KUKA KRL program: MyProgram_169().src

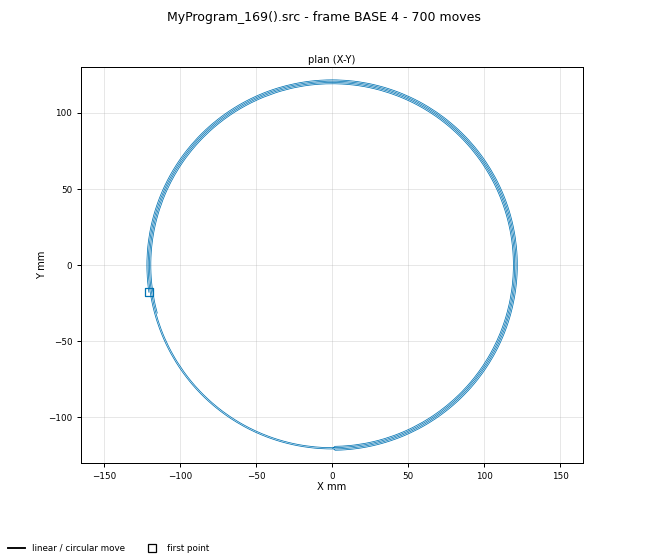
[picture p0: tool path of MyProgram_169().src in frame BASE 4, 700 of 700 moves have a stored position in this frame; points joined in program order, loops and branches not executed]
&ACCESS RVP
&REL 1
&PARAM TEMPLATE = C:\KRC\Roboter\Template\vorgabe
&PARAM EDITMASK = *
DEF MyProgram_169()
; ---- Setting reference (Base) ----
$BASE = BASE_DATA[4]

; --------------------------
; ---- Setting tool (TCP) ----
$TOOL = TOOL_DATA[3]
; --------------------------

$VEL.CP = VEL_APROX_PRINT
Startdeposition()
$VEL.CP = VEL_PRINT
LIN {X -120.4761,Y -17.8709,Z 127,A -175.5982,B 24.9546,C -1.5561,E1 24.8414,E2 261.8458} C_DIS
LIN {X -120.8784,Y -14.9089,Z 127,A -177.0141,B 24.9544,C -1.5602,E1 24.8409,E2 263.2603} C_DIS
LIN {X -121.2969,Y -10.9729,Z 127,A -178.8966,B 24.9541,C -1.5654,E1 24.8404,E2 265.1418} C_DIS
LIN {X -121.5297,Y -7.9928,Z 127,A 179.6363,B 24.954,C -1.5674,E1 24.8401,E2 266.6131} C_DIS
LIN {X -121.7415,Y -3.5142,Z 127,A 177.5701,B 24.9535,C -1.5761,E1 24.8398,E2 268.6709} C_DIS
LIN {X -121.7924,Y -0.3822,Z 127,A 176.0888,B 24.9532,C -1.5805,E1 24.8398,E2 270.1505} C_DIS
LIN {X -121.7576,Y 2.989,Z 127,A 174.4893,B 24.9529,C -1.5851,E1 24.8398,E2 271.7487} C_DIS
LIN {X -121.6476,Y 5.9762,Z 127,A 173.073,B 24.9527,C -1.5893,E1 24.84,E2 273.1637} C_DIS
LIN {X -121.479,Y 8.7426,Z 127,A 171.7841,B 24.9524,C -1.5942,E1 24.8403,E2 274.4485} C_DIS
LIN {X -121.2078,Y 11.9379,Z 127,A 170.241,B 24.9522,C -1.5977,E1 24.8407,E2 275.9927} C_DIS
LIN {X -120.7538,Y 15.8701,Z 127,A 168.3665,B 24.9518,C -1.6032,E1 24.8413,E2 277.8651} C_DIS
LIN {X -120.2477,Y 19.348,Z 127,A 166.7006,B 24.9515,C -1.6081,E1 24.842,E2 279.5294} C_DIS
LIN {X -119.8297,Y 21.776,Z 127,A 165.4749,B 24.9515,C -1.609,E1 24.8426,E2 280.7601} C_DIS
LIN {X -118.947,Y 26.1719,Z 127,A 163.3508,B 24.9511,C -1.6152,E1 24.8438,E2 282.882} C_DIS
LIN {X -118.1443,Y 29.5936,Z 127,A 161.7444,B 24.9507,C -1.6225,E1 24.8448,E2 284.4804} C_DIS
LIN {X -117.1182,Y 33.4165,Z 127,A 159.8693,B 24.9503,C -1.628,E1 24.8462,E2 286.3533} C_DIS
LIN {X -116.1073,Y 36.7826,Z 127,A 158.2044,B 24.95,C -1.6327,E1 24.8476,E2 288.0166} C_DIS
LIN {X -114.8487,Y 40.5354,Z 127,A 156.3297,B 24.9497,C -1.6381,E1 24.8493,E2 289.8892} C_DIS
LIN {X -113.8193,Y 43.3418,Z 127,A 154.914,B 24.9495,C -1.6421,E1 24.8507,E2 291.3033} C_DIS
LIN {X -112.7214,Y 46.122,Z 127,A 153.4984,B 24.9492,C -1.646,E1 24.8521,E2 292.7174} C_DIS
LIN {X -111.5555,Y 48.8744,Z 127,A 152.0828,B 24.949,C -1.65,E1 24.8537,E2 294.1314} C_DIS
LIN {X -110.3225,Y 51.5974,Z 127,A 150.6089,B 24.949,C -1.6514,E1 24.8554,E2 295.6101} C_DIS
LIN {X -108.3486,Y 55.6231,Z 127,A 148.5441,B 24.9484,C -1.6596,E1 24.858,E2 297.6663} C_DIS
LIN {X -106.7004,Y 58.7272,Z 127,A 146.8803,B 24.9481,C -1.664,E1 24.8602,E2 299.3284} C_DIS
LIN {X -104.7338,Y 62.1624,Z 127,A 144.948,B 24.948,C -1.6665,E1 24.8629,E2 301.2648} C_DIS
LIN {X -102.4536,Y 65.8526,Z 127,A 142.9275,B 24.9475,C -1.6732,E1 24.8659,E2 303.2795} C_DIS
LIN {X -100.7249,Y 68.4678,Z 127,A 141.4691,B 24.9472,C -1.6781,E1 24.8681,E2 304.7336} C_DIS
LIN {X -99.0143,Y 70.9191,Z 127,A 140.0543,B 24.947,C -1.6817,E1 24.8704,E2 306.1469} C_DIS
LIN {X -97.244,Y 73.3277,Z 127,A 138.6399,B 24.9468,C -1.6852,E1 24.8728,E2 307.5597} C_DIS
LIN {X -95.4152,Y 75.6921,Z 127,A 137.1671,B 24.9468,C -1.6861,E1 24.8753,E2 309.0373} C_DIS
LIN {X -92.5645,Y 79.1527,Z 127,A 135.1043,B 24.9462,C -1.6936,E1 24.879,E2 311.0916} C_DIS
LIN {X -90.2436,Y 81.7921,Z 127,A 133.4417,B 24.946,C -1.6975,E1 24.8821,E2 312.7526} C_DIS
LIN {X -88.4889,Y 83.6847,Z 127,A 132.2359,B 24.9458,C -1.7009,E1 24.8844,E2 313.9555} C_DIS
LIN {X -86.1216,Y 86.1216,Z 127,A 130.614,B 24.9456,C -1.7038,E1 24.8875,E2 315.5774} C_DIS
LIN {X -83.2761,Y 88.8731,Z 127,A 128.6841,B 24.9455,C -1.7053,E1 24.8915,E2 317.5116} C_DIS
LIN {X -81.07,Y 90.8901,Z 127,A 127.3051,B 24.9452,C -1.7098,E1 24.8943,E2 318.8854} C_DIS
LIN {X -78.415,Y 93.193,Z 127,A 125.6676,B 24.9449,C -1.7142,E1 24.8978,E2 320.5188} C_DIS
LIN {X -75.344,Y 95.6903,Z 127,A 123.7965,B 24.9447,C -1.718,E1 24.9018,E2 322.388} C_DIS
LIN {X -72.9729,Y 97.5105,Z 127,A 122.3839,B 24.9445,C -1.7207,E1 24.905,E2 323.7992} C_DIS
LIN {X -70.5579,Y 99.272,Z 127,A 120.913,B 24.9445,C -1.7207,E1 24.9083,E2 325.2751} C_DIS
LIN {X -67.6653,Y 101.2683,Z 127,A 119.3107,B 24.9442,C -1.7263,E1 24.912,E2 326.8696} C_DIS
LIN {X -64.3377,Y 103.4118,Z 127,A 117.4409,B 24.9439,C -1.7295,E1 24.9164,E2 328.7377} C_DIS
LIN {X -61.7805,Y 104.9596,Z 127,A 116.0291,B 24.9438,C -1.7319,E1 24.9198,E2 330.1482} C_DIS
LIN {X -59.186,Y 106.4442,Z 127,A 114.6303,B 24.9436,C -1.7347,E1 24.9232,E2 331.5444} C_DIS
LIN {X -56.5559,Y 107.8646,Z 127,A 113.2061,B 24.9435,C -1.7363,E1 24.9267,E2 332.9687} C_DIS
LIN {X -53.8918,Y 109.2201,Z 127,A 111.7368,B 24.9435,C -1.7358,E1 24.9304,E2 334.4431} C_DIS
LIN {X -50.7187,Y 110.7315,Z 127,A 110.136,B 24.9432,C -1.7407,E1 24.9344,E2 336.0363} C_DIS
LIN {X -47.986,Y 111.9428,Z 127,A 108.7252,B 24.9431,C -1.7426,E1 24.938,E2 337.446} C_DIS
LIN {X -45.2243,Y 113.0868,Z 127,A 107.3148,B 24.943,C -1.7444,E1 24.9417,E2 338.8552} C_DIS
LIN {X -42.4354,Y 114.1626,Z 127,A 105.9046,B 24.9429,C -1.7461,E1 24.9453,E2 340.2643} C_DIS
LIN {X -38.7026,Y 115.4792,Z 127,A 104.0371,B 24.9427,C -1.7482,E1 24.9503,E2 342.1304} C_DIS
LIN {X -35.355,Y 116.5499,Z 127,A 102.3796,B 24.9427,C -1.7499,E1 24.9547,E2 343.7868} C_DIS
LIN {X -32.4841,Y 117.3824,Z 127,A 100.9703,B 24.9425,C -1.7513,E1 24.9585,E2 345.1949} C_DIS
LIN {X -30.1025,Y 118.0135,Z 127,A 99.8086,B 24.9425,C -1.7524,E1 24.9616,E2 346.3558} C_DIS
LIN {X -27.0068,Y 118.7607,Z 127,A 98.3284,B 24.9423,C -1.7546,E1 24.9656,E2 347.8328} C_DIS
LIN {X -24.2756,Y 119.3484,Z 127,A 96.9905,B 24.9423,C -1.7546,E1 24.9693,E2 349.172} C_DIS
LIN {X -20.8222,Y 120.0012,Z 127,A 95.3345,B 24.9423,C -1.7558,E1 24.9738,E2 350.8271} C_DIS
LIN {X -17.8709,Y 120.4761,Z 127,A 93.9263,B 24.9422,C -1.7567,E1 24.9777,E2 352.2345} C_DIS
LIN {X -14.9089,Y 120.8784,Z 127,A 92.5183,B 24.9422,C -1.7575,E1 24.9816,E2 353.6417} C_DIS
LIN {X -10.9729,Y 121.2969,Z 127,A 90.6182,B 24.9422,C -1.7568,E1 24.9869,E2 355.5445} C_DIS
LIN {X -7.9928,Y 121.5297,Z 127,A 89.1883,B 24.9422,C -1.7563,E1 24.9909,E2 356.976} C_DIS
LIN {X -3.5142,Y 121.7415,Z 127,A 87.1351,B 24.942,C -1.7596,E1 24.9966,E2 359.0219} C_DIS
LIN {X 0,Y 121.7943,Z 127,A 85.4814,B 24.942,C -1.7599,E1 25.0012,E2 360.6749} C_DIS
LIN {X 2.989,Y 121.7576,Z 127,A 84.0744,B 24.942,C -1.76,E1 25.0051,E2 362.0813} C_DIS
LIN {X 5.9762,Y 121.6476,Z 127,A 82.668,B 24.942,C -1.76,E1 25.009,E2 363.4872} C_DIS
LIN {X 8.8861,Y 121.4693,Z 127,A 81.3102,B 24.9419,C -1.7607,E1 25.0128,E2 364.8429} C_DIS
LIN {X 11.9379,Y 121.2078,Z 127,A 79.8563,B 24.9419,C -1.7599,E1 25.0169,E2 366.2978} C_DIS
LIN {X 14.387,Y 120.9395,Z 127,A 78.6973,B 24.9419,C -1.7598,E1 25.0201,E2 367.4564} C_DIS
LIN {X 17.3507,Y 120.55,Z 127,A 77.2919,B 24.9419,C -1.7595,E1 25.024,E2 368.8613} C_DIS
LIN {X 20.5987,Y 120.0386,Z 127,A 75.7701,B 24.9419,C -1.7601,E1 25.0281,E2 370.3801} C_DIS
LIN {X 23.2449,Y 119.5534,Z 127,A 74.4816,B 24.942,C -1.7585,E1 25.0317,E2 371.6708} C_DIS
LIN {X 26.6853,Y 118.835,Z 127,A 72.8298,B 24.942,C -1.7577,E1 25.0362,E2 373.3223} C_DIS
LIN {X 30.5323,Y 117.903,Z 127,A 70.97,B 24.9422,C -1.7568,E1 25.0412,E2 375.1816} C_DIS
LIN {X 33.4165,Y 117.1182,Z 127,A 69.566,B 24.9422,C -1.7559,E1 25.045,E2 376.5855} C_DIS
LIN {X 36.7826,Y 116.1072,Z 127,A 67.9153,B 24.9422,C -1.7547,E1 25.0494,E2 378.2359} C_DIS
LIN {X 40.5354,Y 114.8487,Z 127,A 66.0565,B 24.9424,C -1.7533,E1 25.0543,E2 380.0945} C_DIS
LIN {X 43.3418,Y 113.8193,Z 127,A 64.6532,B 24.9424,C -1.7521,E1 25.058,E2 381.4977} C_DIS
LIN {X 46.122,Y 112.7214,Z 127,A 63.1921,B 24.9427,C -1.748,E1 25.0618,E2 382.965} C_DIS
LIN {X 49.0979,Y 111.4581,Z 127,A 61.7559,B 24.9426,C -1.7503,E1 25.0655,E2 384.3923} C_DIS
LIN {X 51.5974,Y 110.3225,Z 127,A 60.3866,B 24.9429,C -1.7451,E1 25.069,E2 385.7705} C_DIS
LIN {X 54.2893,Y 109.023,Z 127,A 58.9841,B 24.943,C -1.7435,E1 25.0725,E2 387.173} C_DIS
LIN {X 57.3868,Y 107.427,Z 127,A 57.4071,B 24.943,C -1.7443,E1 25.0764,E2 388.744} C_DIS
LIN {X 60.0322,Y 105.9716,Z 127,A 55.9912,B 24.943,C -1.7425,E1 25.0798,E2 390.1599} C_DIS
LIN {X 63.443,Y 103.9631,Z 127,A 54.135,B 24.9433,C -1.74,E1 25.0843,E2 392.0163} C_DIS
LIN {X 66.4175,Y 102.091,Z 127,A 52.4873,B 24.9434,C -1.7376,E1 25.0881,E2 393.6643} C_DIS
LIN {X 68.4678,Y 100.7249,Z 127,A 51.3323,B 24.9435,C -1.7359,E1 25.0908,E2 394.8194} C_DIS
LIN {X 71.3468,Y 98.7091,Z 127,A 49.6849,B 24.9437,C -1.7333,E1 25.0946,E2 396.4672} C_DIS
LIN {X 73.3277,Y 97.244,Z 127,A 48.4725,B 24.944,C -1.7287,E1 25.0973,E2 397.6862} C_DIS
LIN {X 76.1043,Y 95.0893,Z 127,A 46.8832,B 24.944,C -1.7287,E1 25.1008,E2 399.2696} C_DIS
LIN {X 78.415,Y 93.193,Z 127,A 45.4829,B 24.9442,C -1.7262,E1 25.1038,E2 400.6703} C_DIS
LIN {X 80.4881,Y 91.4068,Z 127,A 44.2246,B 24.9442,C -1.7251,E1 25.1064,E2 401.9263} C_DIS
LIN {X 82.8933,Y 89.2331,Z 127,A 42.6826,B 24.9445,C -1.7211,E1 25.1096,E2 403.4715} C_DIS
LIN {X 85.0583,Y 87.1719,Z 127,A 41.283,B 24.9447,C -1.7184,E1 25.1124,E2 404.8716} C_DIS
LIN {X 88.2092,Y 83.9821,Z 127,A 39.1831,B 24.9449,C -1.7142,E1 25.1165,E2 406.9724} C_DIS
LIN {X 90.1788,Y 81.8627,Z 127,A 37.8259,B 24.9451,C -1.7113,E1 25.1191,E2 408.3304} C_DIS
LIN {X 92.2237,Y 79.5527,Z 127,A 36.3843,B 24.9453,C -1.7084,E1 25.1217,E2 409.7724} C_DIS
LIN {X 93.9,Y 77.5642,Z 127,A 35.1835,B 24.9454,C -1.7066,E1 25.1239,E2 410.9719} C_DIS
LIN {X 96.0161,Y 74.9317,Z 127,A 33.5862,B 24.9457,C -1.7023,E1 25.1267,E2 412.5718} C_DIS
LIN {X 97.8261,Y 72.5528,Z 127,A 32.1876,B 24.9459,C -1.6992,E1 25.129,E2 413.9712} C_DIS
LIN {X 99.5772,Y 70.1302,Z 127,A 30.7889,B 24.9461,C -1.696,E1 25.1313,E2 415.3707} C_DIS
LIN {X 101.2683,Y 67.6653,Z 127,A 29.3903,B 24.9463,C -1.6927,E1 25.1335,E2 416.77} C_DIS
LIN {X 102.8984,Y 65.1597,Z 127,A 27.9919,B 24.9465,C -1.6894,E1 25.1356,E2 418.1694} C_DIS
LIN {X 104.1936,Y 63.0638,Z 127,A 26.8099,B 24.9468,C -1.6852,E1 25.1373,E2 419.3552} C_DIS
LIN {X 105.9716,Y 60.0322,Z 127,A 25.1958,B 24.9469,C -1.6826,E1 25.1396,E2 420.9672} C_DIS
LIN {X 107.1624,Y 57.8753,Z 127,A 23.9859,B 24.9473,C -1.6769,E1 25.1412,E2 422.1841} C_DIS
LIN {X 108.7896,Y 54.7601,Z 127,A 22.4,B 24.9473,C -1.6755,E1 25.1432,E2 423.7648} C_DIS
LIN {X 110.5097,Y 51.1951,Z 127,A 20.549,B 24.9477,C -1.6708,E1 25.1454,E2 425.617} C_DIS
LIN {X 111.9428,Y 47.986,Z 127,A 18.9056,B 24.948,C -1.6664,E1 25.1473,E2 427.2618} C_DIS
LIN {X 113.0047,Y 45.4259,Z 127,A 17.6339,B 24.9481,C -1.6642,E1 25.1486,E2 428.5317} C_DIS
LIN {X 114.1626,Y 42.4354,Z 127,A 16.1111,B 24.9484,C -1.659,E1 25.1501,E2 430.0583} C_DIS
LIN {X 115.4792,Y 38.7026,Z 127,A 14.2361,B 24.9488,C -1.6527,E1 25.1519,E2 431.9375} C_DIS
LIN {X 116.5499,Y 35.355,Z 127,A 12.618,B 24.949,C -1.6494,E1 25.1532,E2 433.5543} C_DIS
LIN {X 117.3824,Y 32.4841,Z 127,A 11.2212,B 24.9493,C -1.6455,E1 25.1543,E2 434.9522} C_DIS
LIN {X 118.374,Y 28.6521,Z 127,A 9.3711,B 24.9496,C -1.6403,E1 25.1555,E2 436.8038} C_DIS
LIN {X 119.1535,Y 25.225,Z 127,A 7.7291,B 24.9499,C -1.6356,E1 25.1565,E2 438.4474} C_DIS
LIN {X 120.0012,Y 20.8222,Z 127,A 5.6337,B 24.9502,C -1.6296,E1 25.1576,E2 440.5447} C_DIS
LIN {X 120.4761,Y 17.8709,Z 127,A 4.2371,B 24.9505,C -1.6256,E1 25.1582,E2 441.9425} C_DIS
LIN {X 120.8784,Y 14.9089,Z 127,A 2.8405,B 24.9507,C -1.6216,E1 25.1587,E2 443.3404} C_DIS
LIN {X 121.1531,Y 12.4605,Z 127,A 1.6525,B 24.951,C -1.6164,E1 25.1591,E2 444.5336} C_DIS
LIN {X 121.4643,Y 8.9597,Z 127,A 0.047,B 24.9512,C -1.6134,E1 25.1594,E2 446.1366} C_DIS
LIN {X 121.6476,Y 5.9762,Z 127,A -1.3495,B 24.9515,C -1.6093,E1 25.1596,E2 447.5344} C_DIS
LIN {X 121.7576,Y 2.989,Z 127,A -2.746,B 24.9517,C -1.6052,E1 25.1598,E2 448.9323} C_DIS
LIN {X 121.7924,Y -0.3822,Z 127,A -4.1792,B 24.9516,C -1.6077,E1 25.1598,E2 450.3511} C_DIS
LIN {X 121.7576,Y -2.989,Z 127,A -5.5389,B 24.9522,C -1.597,E1 25.1598,E2 451.728} C_DIS
LIN {X 121.6476,Y -5.9762,Z 127,A -6.9354,B 24.9525,C -1.5928,E1 25.1595,E2 453.126} C_DIS
LIN {X 121.4643,Y -8.9597,Z 127,A -8.3318,B 24.9527,C -1.5887,E1 25.1593,E2 454.5238} C_DIS
LIN {X 121.2078,Y -11.9379,Z 127,A -9.728,B 24.953,C -1.5846,E1 25.1589,E2 455.9215} C_DIS
LIN {X 120.7538,Y -15.8701,Z 127,A -11.6351,B 24.9534,C -1.5763,E1 25.1583,E2 457.8368} C_DIS
LIN {X 120.328,Y -18.8287,Z 127,A -13.0315,B 24.9537,C -1.5722,E1 25.1577,E2 459.2347} C_DIS
LIN {X 119.8297,Y -21.776,Z 127,A -14.428,B 24.9539,C -1.5681,E1 25.157,E2 460.6327} C_DIS
LIN {X 119.2217,Y -24.8928,Z 127,A -15.8805,B 24.9541,C -1.5653,E1 25.1562,E2 462.0833} C_DIS
LIN {X 118.6168,Y -27.6296,Z 127,A -17.2211,B 24.9544,C -1.5599,E1 25.1554,E2 463.4288} C_DIS
LIN {X 117.5195,Y -31.9768,Z 127,A -19.2586,B 24.9546,C -1.5567,E1 25.154,E2 465.4621} C_DIS
LIN {X 116.6993,Y -34.8513,Z 127,A -20.6555,B 24.9548,C -1.5527,E1 25.1529,E2 466.8605} C_DIS
LIN {X 115.8089,Y -37.7047,Z 127,A -22.1095,B 24.9552,C -1.5458,E1 25.1516,E2 468.3225} C_DIS
LIN {X 114.6747,Y -41.0313,Z 127,A -23.6945,B 24.9553,C -1.5439,E1 25.1502,E2 469.903} C_DIS
LIN {X 113.1249,Y -45.1272,Z 127,A -25.7238,B 24.9556,C -1.539,E1 25.1481,E2 471.9325} C_DIS
LIN {X 112.1469,Y -47.5018,Z 127,A -26.9413,B 24.9559,C -1.5348,E1 25.1468,E2 473.1532} C_DIS
LIN {X 110.7315,Y -50.7188,Z 127,A -28.5838,B 24.9561,C -1.5302,E1 25.1449,E2 474.7976} C_DIS
LIN {X 109.023,Y -54.2893,Z 127,A -30.4342,B 24.9564,C -1.5252,E1 25.1427,E2 476.65} C_DIS
LIN {X 107.413,Y -57.4134,Z 127,A -32.0769,B 24.9567,C -1.5207,E1 25.1406,E2 478.2945} C_DIS
LIN {X 105.9716,Y -60.0322,Z 127,A -33.4742,B 24.9569,C -1.517,E1 25.1387,E2 479.6934} C_DIS
LIN {X 104.4665,Y -62.6148,Z 127,A -34.8717,B 24.9571,C -1.5133,E1 25.1367,E2 481.0924} C_DIS
LIN {X 103.1304,Y -64.7883,Z 127,A -36.1065,B 24.9574,C -1.5081,E1 25.1348,E2 482.3331} C_DIS
LIN {X 100.7249,Y -68.4678,Z 127,A -38.1778,B 24.9577,C -1.5021,E1 25.1316,E2 484.4084} C_DIS
LIN {X 98.7091,Y -71.3468,Z 127,A -39.7641,B 24.9578,C -1.5007,E1 25.1291,E2 485.9901} C_DIS
LIN {X 96.0161,Y -74.9317,Z 127,A -41.861,B 24.9581,C -1.4956,E1 25.1255,E2 488.0893} C_DIS
LIN {X 94.1483,Y -77.2655,Z 127,A -43.2591,B 24.9583,C -1.4922,E1 25.1231,E2 489.4888} C_DIS
LIN {X 91.5862,Y -80.2827,Z 127,A -45.1686,B 24.9587,C -1.485,E1 25.1196,E2 491.4067} C_DIS
LIN {X 89.5884,Y -82.5062,Z 127,A -46.5672,B 24.9589,C -1.4817,E1 25.1169,E2 492.8068} C_DIS
LIN {X 86.4909,Y -85.7477,Z 127,A -48.6653,B 24.9591,C -1.477,E1 25.1129,E2 494.907} C_DIS
LIN {X 83.9821,Y -88.2092,Z 127,A -50.2525,B 24.9591,C -1.4762,E1 25.1097,E2 496.4895} C_DIS
LIN {X 81.7921,Y -90.2436,Z 127,A -51.6517,B 24.9593,C -1.4732,E1 25.1068,E2 497.8902} C_DIS
LIN {X 79.5527,Y -92.2237,Z 127,A -53.0511,B 24.9595,C -1.4702,E1 25.1039,E2 499.2909} C_DIS
LIN {X 76.5182,Y -94.7539,Z 127,A -54.902,B 24.9597,C -1.4665,E1 25.0999,E2 501.1437} C_DIS
LIN {X 74.164,Y -96.6077,Z 127,A -56.3617,B 24.96,C -1.4609,E1 25.0966,E2 502.6111} C_DIS
LIN {X 71.3468,Y -98.7091,Z 127,A -57.9498,B 24.96,C -1.4606,E1 25.0931,E2 504.1944} C_DIS
LIN {X 67.6925,Y -101.2499,Z 127,A -60.0261,B 24.9602,C -1.4571,E1 25.0883,E2 506.2717} C_DIS
LIN {X 64.3377,Y -103.4118,Z 127,A -61.9047,B 24.9604,C -1.4535,E1 25.0839,E2 508.1529} C_DIS
LIN {X 61.7805,Y -104.9596,Z 127,A -63.3053,B 24.9606,C -1.4511,E1 25.0805,E2 509.5548} C_DIS
LIN {X 59.186,Y -106.4442,Z 127,A -64.7638,B 24.9608,C -1.446,E1 25.0769,E2 511.021} C_DIS
LIN {X 56.5559,Y -107.8646,Z 127,A -66.1647,B 24.9609,C -1.4438,E1 25.0735,E2 512.4231} C_DIS
LIN {X 53.421,Y -109.4534,Z 127,A -67.7546,B 24.9609,C -1.4441,E1 25.0695,E2 514.008} C_DIS
LIN {X 51.1951,Y -110.5097,Z 127,A -68.9098,B 24.961,C -1.4425,E1 25.0666,E2 515.1641} C_DIS
LIN {X 47.986,Y -111.9428,Z 127,A -70.5579,B 24.9611,C -1.4402,E1 25.0624,E2 516.8137} C_DIS
LIN {X 45.3148,Y -113.0499,Z 127,A -71.8974,B 24.9611,C -1.4392,E1 25.0589,E2 518.1523} C_DIS
LIN {X 42.4354,Y -114.1626,Z 127,A -73.3617,B 24.9613,C -1.4366,E1 25.0551,E2 519.6197} C_DIS
LIN {X 38.7026,Y -115.4792,Z 127,A -75.2768,B 24.9616,C -1.4317,E1 25.05,E2 521.5426} C_DIS
LIN {X 35.355,Y -116.5499,Z 127,A -76.8683,B 24.9616,C -1.4326,E1 25.0458,E2 523.1289} C_DIS
LIN {X 32.4841,Y -117.3824,Z 127,A -78.271,B 24.9616,C -1.4312,E1 25.042,E2 524.5326} C_DIS
LIN {X 29.5936,Y -118.1443,Z 127,A -79.6742,B 24.9616,C -1.4299,E1 25.0382,E2 525.9368} C_DIS
LIN {X 26.6853,Y -118.835,Z 127,A -81.0777,B 24.9618,C -1.4287,E1 25.0344,E2 527.3412} C_DIS
LIN {X 22.8092,Y -119.6373,Z 127,A -82.9731,B 24.9619,C -1.4255,E1 25.0292,E2 529.2419} C_DIS
LIN {X 19.8663,Y -120.161,Z 127,A -84.3981,B 24.962,C -1.4235,E1 25.0253,E2 530.6701} C_DIS
LIN {X 16.9114,Y -120.6124,Z 127,A -85.8021,B 24.962,C -1.4226,E1 25.0214,E2 532.075} C_DIS
LIN {X 13.4321,Y -121.0513,Z 127,A -87.3904,B 24.962,C -1.4245,E1 25.017,E2 533.6576} C_DIS
LIN {X 8.9597,Y -121.4643,Z 127,A -89.5027,B 24.962,C -1.4234,E1 25.0111,E2 535.7713} C_DIS
LIN {X 5.9762,Y -121.6476,Z 127,A -90.9077,B 24.962,C -1.4229,E1 25.0072,E2 537.177} C_DIS
LIN {X 2.02,Y -121.7755,Z 127,A -92.7723,B 24.9621,C -1.4222,E1 25.002,E2 539.0428} C_DIS
LIN {X 2.02,Y -121.7755,Z 127,A -92.7723,B 24.9621,C -1.4222,E1 25.002,E2 539.0428} C_DIS
Enddeposition()
LIN {X 0.8498,Y -120.9267,Z 127,A -92.499,B 24.9592,C -1.476,E1 25.0031,E2 538.6421} C_DIS
Startdeposition()
$VEL.CP = VEL_PRINT
LIN {X 6.1613,Y -120.7806,Z 127,A -89.7657,B 24.9586,C -1.4871,E1 25.0108,E2 535.8835} C_DIS
LIN {X 9.6002,Y -120.5549,Z 127,A -88.5598,B 24.9597,C -1.4675,E1 25.014,E2 534.7243} C_DIS
LIN {X 12.7244,Y -120.2653,Z 127,A -87.0113,B 24.9594,C -1.4713,E1 25.0183,E2 533.168} C_DIS
LIN {X 17.3332,Y -119.6884,Z 127,A -84.2229,B 24.9578,C -1.501,E1 25.0263,E2 530.3116} C_DIS
LIN {X 21.9078,Y -118.9368,Z 127,A -82.5343,B 24.9591,C -1.4783,E1 25.0307,E2 528.6786} C_DIS
LIN {X 25.5115,Y -118.2154,Z 127,A -80.9082,B 24.9593,C -1.4744,E1 25.0352,E2 527.0639} C_DIS
LIN {X 28.6124,Y -117.5031,Z 127,A -79.4189,B 24.9593,C -1.475,E1 25.0392,E2 525.5753} C_DIS
LIN {X 32.2121,Y -116.5698,Z 127,A -77.5756,B 24.9589,C -1.4807,E1 25.0442,E2 523.7212} C_DIS
LIN {X 35.1312,Y -115.7236,Z 127,A -75.4821,B 24.957,C -1.5142,E1 25.05,E2 521.5524} C_DIS
LIN {X 39.9144,Y -114.16,Z 127,A -73.194,B 24.9571,C -1.5126,E1 25.056,E2 519.2726} C_DIS
LIN {X 44.3276,Y -112.5199,Z 127,A -71.8403,B 24.9594,C -1.473,E1 25.0593,E2 518.0154} C_DIS
LIN {X 47.9828,Y -111.011,Z 127,A -69.6996,B 24.9585,C -1.4887,E1 25.0649,E2 515.8427} C_DIS
LIN {X 51.186,Y -109.5704,Z 127,A -68.0535,B 24.9584,C -1.4905,E1 25.069,E2 514.1965} C_DIS
LIN {X 54.5225,Y -107.9503,Z 127,A -66.317,B 24.9583,C -1.4924,E1 25.0734,E2 512.4602} C_DIS
LIN {X 58.0159,Y -106.1129,Z 127,A -64.4585,B 24.9581,C -1.4951,E1 25.078,E2 510.6006} C_DIS
LIN {X 61.2525,Y -104.2779,Z 127,A -62.6716,B 24.9579,C -1.4995,E1 25.0823,E2 508.8086} C_DIS
LIN {X 64.1573,Y -102.5158,Z 127,A -61.0731,B 24.9577,C -1.5021,E1 25.0861,E2 507.2092} C_DIS
LIN {X 67.5687,Y -100.3005,Z 127,A -59.3271,B 24.958,C -1.497,E1 25.0901,E2 505.4808} C_DIS
LIN {X 72.1717,Y -97.0424,Z 127,A -56.1531,B 24.9563,C -1.5273,E1 25.0975,E2 502.2464} C_DIS
LIN {X 74.8604,Y -94.982,Z 127,A -54.9366,B 24.9572,C -1.5117,E1 25.1,E2 501.0714} C_DIS
LIN {X 79.4487,Y -91.1788,Z 127,A -52.0227,B 24.9566,C -1.5226,E1 25.1063,E2 498.143} C_DIS
LIN {X 82.7863,Y -88.1594,Z 127,A -49.946,B 24.9564,C -1.5249,E1 25.1105,E2 496.0692} C_DIS
LIN {X 86.0248,Y -85.0023,Z 127,A -47.4355,B 24.9551,C -1.5485,E1 25.1156,E2 493.5136} C_DIS
LIN {X 88.6717,Y -82.2391,Z 127,A -45.9364,B 24.9557,C -1.5375,E1 25.1184,E2 492.0473} C_DIS
LIN {X 93.5426,Y -76.6541,Z 127,A -42.6577,B 24.9558,C -1.5351,E1 25.1243,E2 488.789} C_DIS
LIN {X 97.9667,Y -70.9126,Z 127,A -39.0659,B 24.9549,C -1.5523,E1 25.1304,E2 485.1736} C_DIS
LIN {X 100.0389,Y -67.9551,Z 127,A -37.4767,B 24.9549,C -1.5511,E1 25.1329,E2 483.5951} C_DIS
LIN {X 101.5025,Y -65.7505,Z 127,A -36.05,B 24.9542,C -1.5633,E1 25.1351,E2 482.1468} C_DIS
LIN {X 103.9195,Y -61.8589,Z 127,A -34.0196,B 24.9542,C -1.5626,E1 25.1381,E2 480.1283} C_DIS
LIN {X 106.0589,Y -58.1155,Z 127,A -31.8672,B 24.9536,C -1.5742,E1 25.141,E2 477.9599} C_DIS
LIN {X 108.128,Y -54.1687,Z 127,A -29.947,B 24.9538,C -1.571,E1 25.1434,E2 476.0575} C_DIS
LIN {X 109.5966,Y -51.1295,Z 127,A -27.6686,B 24.9514,C -1.6101,E1 25.1462,E2 473.6991} C_DIS
LIN {X 111.5748,Y -46.6565,Z 127,A -25.9265,B 24.9527,C -1.5882,E1 25.1481,E2 472.0181} C_DIS
LIN {X 112.8287,Y -43.5406,Z 127,A -24.3633,B 24.9525,C -1.5918,E1 25.1496,E2 470.4552} C_DIS
LIN {X 114.2091,Y -39.7745,Z 127,A -22.5326,B 24.9524,C -1.5943,E1 25.1514,E2 468.6289} C_DIS
LIN {X 115.4976,Y -35.8602,Z 127,A -20.7468,B 24.9525,C -1.5921,E1 25.1529,E2 466.8583} C_DIS
LIN {X 116.2006,Y -33.517,Z 127,A -19.5938,B 24.9523,C -1.5955,E1 25.1538,E2 465.7038} C_DIS
LIN {X 117.0607,Y -30.373,Z 127,A -17.9082,B 24.9516,C -1.6076,E1 25.155,E2 463.9995} C_DIS
LIN {X 118.0996,Y -26.0426,Z 127,A -15.8721,B 24.9514,C -1.6107,E1 25.1563,E2 461.9678} C_DIS
LIN {X 118.6259,Y -23.5373,Z 127,A -14.12,B 24.9495,C -1.6419,E1 25.1573,E2 460.1525} C_DIS
LIN {X 119.3576,Y -19.4841,Z 127,A -11.8288,B 24.948,C -1.6655,E1 25.1583,E2 457.819} C_DIS
LIN {X 120.1583,Y -13.7026,Z 127,A -10.204,B 24.951,C -1.6169,E1 25.1588,E2 456.3184} C_DIS
LIN {X 120.6907,Y -7.719,Z 127,A -7.1986,B 24.95,C -1.6342,E1 25.1595,E2 453.2902} C_DIS
LIN {X 120.9156,Y -2.2507,Z 127,A -4.5831,B 24.9494,C -1.6438,E1 25.1598,E2 450.6676} C_DIS
LIN {X 120.9326,Y 1.0405,Z 127,A -2.6111,B 24.9478,C -1.6697,E1 25.1598,E2 448.6463} C_DIS
LIN {X 120.8476,Y 4.667,Z 127,A -1.4404,B 24.9491,C -1.6477,E1 25.1596,E2 447.5344} C_DIS
LIN {X 120.5298,Y 9.9136,Z 127,A 1.0724,B 24.9486,C -1.6569,E1 25.1592,E2 445.0148} C_DIS
LIN {X 119.835,Y 16.3014,Z 127,A 4.1713,B 24.9478,C -1.6694,E1 25.1582,E2 441.9049} C_DIS
LIN {X 119.3699,Y 19.4104,Z 127,A 5.7343,B 24.9472,C -1.6778,E1 25.1575,E2 440.3311} C_DIS
LIN {X 118.7629,Y 22.8257,Z 127,A 7.3217,B 24.9471,C -1.6803,E1 25.1567,E2 438.7472} C_DIS
LIN {X 117.9466,Y 26.7299,Z 127,A 9.2263,B 24.9467,C -1.6869,E1 25.1556,E2 436.8379} C_DIS
LIN {X 117.1848,Y 29.8899,Z 127,A 10.7456,B 24.9464,C -1.6907,E1 25.1545,E2 435.3185} C_DIS
LIN {X 116.1336,Y 33.7502,Z 127,A 12.6999,B 24.9459,C -1.6995,E1 25.153,E2 433.3547} C_DIS
LIN {X 115.0004,Y 37.4246,Z 127,A 14.4424,B 24.9458,C -1.7011,E1 25.1516,E2 431.6182} C_DIS
LIN {X 113.6967,Y 41.2159,Z 127,A 16.6118,B 24.9445,C -1.7203,E1 25.1495,E2 429.4158} C_DIS
LIN {X 111.8909,Y 45.8932,Z 127,A 18.6954,B 24.945,C -1.7128,E1 25.1474,E2 427.3614} C_DIS
LIN {X 110.4039,Y 49.3635,Z 127,A 20.411,B 24.945,C -1.7144,E1 25.1455,E2 425.6515} C_DIS
LIN {X 109.2523,Y 51.8642,Z 127,A 21.8103,B 24.9444,C -1.7228,E1 25.1438,E2 424.2398} C_DIS
LIN {X 107.7678,Y 54.8796,Z 127,A 23.3515,B 24.9442,C -1.7248,E1 25.1419,E2 422.7021} C_DIS
LIN {X 106.0644,Y 58.1054,Z 127,A 25.0874,B 24.9439,C -1.73,E1 25.1396,E2 420.9631} C_DIS
LIN {X 104.2158,Y 61.3576,Z 127,A 26.7893,B 24.9439,C -1.7314,E1 25.1372,E2 419.2668} C_DIS
LIN {X 102.089,Y 64.8369,Z 127,A 28.7704,B 24.9433,C -1.7389,E1 25.1343,E2 417.2779} C_DIS
LIN {X 100.502,Y 67.2711,Z 127,A 30.1844,B 24.943,C -1.7443,E1 25.1321,E2 415.8581} C_DIS
LIN {X 98.455,Y 70.2301,Z 127,A 31.6473,B 24.9435,C -1.7368,E1 25.1298,E2 414.4201} C_DIS
LIN {X 97.0709,Y 72.1337,Z 127,A 32.9753,B 24.9426,C -1.7501,E1 25.1275,E2 413.0672} C_DIS
LIN {X 94.663,Y 75.264,Z 127,A 34.7079,B 24.9427,C -1.7479,E1 25.1246,E2 411.348} C_DIS
LIN {X 92.3646,Y 78.0682,Z 127,A 36.3955,B 24.9426,C -1.7505,E1 25.1215,E2 409.662} C_DIS
LIN {X 90.1956,Y 80.5632,Z 127,A 37.9504,B 24.9424,C -1.7536,E1 25.1187,E2 408.1067} C_DIS
LIN {X 88.5364,Y 82.3854,Z 127,A 39.288,B 24.9416,C -1.7645,E1 25.1161,E2 406.7493} C_DIS
LIN {X 85.9766,Y 85.051,Z 127,A 40.9605,B 24.9416,C -1.7645,E1 25.1128,E2 405.0838} C_DIS
LIN {X 83.1235,Y 87.8423,Z 127,A 42.6587,B 24.942,C -1.7592,E1 25.1095,E2 403.4054} C_DIS
LIN {X 80.9968,Y 89.8073,Z 127,A 44.1581,B 24.9414,C -1.7682,E1 25.1064,E2 401.8907} C_DIS
LIN {X 78.6782,Y 91.8449,Z 127,A 45.599,B 24.9413,C -1.77,E1 25.1033,E2 400.4511} C_DIS
LIN {X 76.6329,Y 93.5598,Z 127,A 46.9868,B 24.9407,C -1.7784,E1 25.1003,E2 399.0488} C_DIS
LIN {X 73.8027,Y 95.8061,Z 127,A 48.5642,B 24.9409,C -1.7751,E1 25.0969,E2 397.485} C_DIS
LIN {X 70.9675,Y 97.9266,Z 127,A 50.2179,B 24.9409,C -1.7769,E1 25.0931,E2 395.8329} C_DIS
LIN {X 67.925,Y 100.0593,Z 127,A 52.1049,B 24.9402,C -1.786,E1 25.0888,E2 393.9309} C_DIS
LIN {X 64.2994,Y 102.427,Z 127,A 54.2022,B 24.9398,C -1.7915,E1 25.0838,E2 391.8275} C_DIS
LIN {X 60.2122,Y 104.8815,Z 127,A 56.4074,B 24.9398,C -1.7923,E1 25.0785,E2 389.6272} C_DIS
LIN {X 56.6016,Y 106.8737,Z 127,A 58.1264,B 24.9404,C -1.7838,E1 25.0744,E2 387.9332} C_DIS
LIN {X 53.9827,Y 108.2201,Z 127,A 59.7187,B 24.9396,C -1.795,E1 25.0703,E2 386.3188} C_DIS
LIN {X 50.3391,Y 109.9642,Z 127,A 61.7007,B 24.9392,C -1.8005,E1 25.0653,E2 384.3287} C_DIS
LIN {X 47.5957,Y 111.1789,Z 127,A 63.2415,B 24.9387,C -1.8078,E1 25.0613,E2 382.7745} C_DIS
LIN {X 43.7491,Y 112.7471,Z 127,A 64.9546,B 24.9394,C -1.7977,E1 25.0569,E2 381.0891} C_DIS
LIN {X 40.1869,Y 114.0643,Z 127,A 66.7141,B 24.9394,C -1.7975,E1 25.0523,E2 379.3337} C_DIS
LIN {X 37.2453,Y 115.0584,Z 127,A 68.179,B 24.9394,C -1.7984,E1 25.0484,E2 377.8694} C_DIS
LIN {X 33.468,Y 116.2145,Z 127,A 70.1224,B 24.9391,C -1.8032,E1 25.0432,E2 375.9181} C_DIS
LIN {X 30.0427,Y 117.1456,Z 127,A 71.7414,B 24.9391,C -1.8013,E1 25.0389,E2 374.306} C_DIS
LIN {X 26.4728,Y 118.0057,Z 127,A 73.585,B 24.9388,C -1.8071,E1 25.0338,E2 372.4512} C_DIS
LIN {X 23.0384,Y 118.722,Z 127,A 75.1383,B 24.9391,C -1.8028,E1 25.0296,E2 370.9101} C_DIS
LIN {X 19.8165,Y 119.302,Z 127,A 76.6984,B 24.9391,C -1.8038,E1 25.0253,E2 369.3492} C_DIS
LIN {X 15.97,Y 119.8782,Z 127,A 78.4708,B 24.9392,C -1.801,E1 25.0204,E2 367.585} C_DIS
LIN {X 9.6785,Y 120.5486,Z 127,A 81.3504,B 24.9395,C -1.7959,E1 25.0125,E2 364.7194} C_DIS
LIN {X 3.0343,Y 120.9003,Z 127,A 85.5678,B 24.9362,C -1.8451,E1 25.0004,E2 360.3864} C_DIS
LIN {X -2.7347,Y 120.9067,Z 127,A 87.2646,B 24.9395,C -1.7964,E1 24.996,E2 358.8049} C_DIS
LIN {X -9.5192,Y 120.5614,Z 127,A 91.6154,B 24.936,C -1.8473,E1 24.9835,E2 354.3319} C_DIS
LIN {X -15.7161,Y 119.9111,Z 127,A 93.543,B 24.9394,C -1.7984,E1 24.9785,E2 352.519} C_DIS
LIN {X -19.3379,Y 119.382,Z 127,A 95.2416,B 24.9396,C -1.7956,E1 24.9738,E2 350.8256} C_DIS
LIN {X -22.6027,Y 118.8059,Z 127,A 96.9772,B 24.9391,C -1.8019,E1 24.969,E2 349.0734} C_DIS
LIN {X -26.5397,Y 117.9906,Z 127,A 98.864,B 24.9393,C -1.7993,E1 24.9639,E2 347.1903} C_DIS
LIN {X -30.0117,Y 117.1535,Z 127,A 100.5008,B 24.9396,C -1.7952,E1 24.9594,E2 345.5609} C_DIS
LIN {X -33.0344,Y 116.3373,Z 127,A 102.0984,B 24.9394,C -1.7988,E1 24.9551,E2 343.9524} C_DIS
LIN {X -37.0774,Y 115.1127,Z 127,A 104.0442,B 24.9397,C -1.794,E1 24.9499,E2 342.0146} C_DIS
LIN {X -41.0063,Y 113.7732,Z 127,A 105.9677,B 24.94,C -1.7895,E1 24.9449,E2 340.0978} C_DIS
LIN {X -45.4273,Y 112.0805,Z 127,A 108.2574,B 24.94,C -1.7886,E1 24.9389,E2 337.8055} C_DIS
LIN {X -48.5043,Y 110.7836,Z 127,A 109.8855,B 24.94,C -1.7883,E1 24.9348,E2 336.1743} C_DIS
LIN {X -52.1558,Y 109.1122,Z 127,A 111.6745,B 24.9406,C -1.7803,E1 24.9303,E2 334.3998} C_DIS
LIN {X -54.7166,Y 107.8511,Z 127,A 113.092,B 24.9406,C -1.781,E1 24.9267,E2 332.977} C_DIS
LIN {X -57.6486,Y 106.3122,Z 127,A 114.6574,B 24.9407,C -1.7781,E1 24.9229,E2 331.4139} C_DIS
LIN {X -60.9415,Y 104.4618,Z 127,A 116.7107,B 24.9402,C -1.7866,E1 24.9178,E2 329.3344} C_DIS
LIN {X -65.1983,Y 101.857,Z 127,A 118.8485,B 24.9411,C -1.7721,E1 24.9128,E2 327.2244} C_DIS
LIN {X -67.9625,Y 100.0339,Z 127,A 120.6368,B 24.9407,C -1.7787,E1 24.9086,E2 325.4144} C_DIS
LIN {X -71.7394,Y 97.3614,Z 127,A 122.6236,B 24.9416,C -1.7651,E1 24.9042,E2 323.453} C_DIS
LIN {X -74.421,Y 95.3293,Z 127,A 124.3751,B 24.9414,C -1.7685,E1 24.9003,E2 321.687} C_DIS
LIN {X -77.6218,Y 92.7399,Z 127,A 126.1945,B 24.942,C -1.7584,E1 24.8964,E2 319.8846} C_DIS
LIN {X -80.4222,Y 90.3217,Z 127,A 128.027,B 24.942,C -1.7579,E1 24.8926,E2 318.0462} C_DIS
LIN {X -83.3447,Y 87.6343,Z 127,A 129.8636,B 24.9425,C -1.7515,E1 24.8888,E2 316.2174} C_DIS
LIN {X -85.7843,Y 85.2457,Z 127,A 131.4557,B 24.9428,C -1.7464,E1 24.8857,E2 314.6306} C_DIS
LIN {X -88.5346,Y 82.3873,Z 127,A 133.4588,B 24.9428,C -1.7471,E1 24.8818,E2 312.6172} C_DIS
LIN {X -90.875,Y 79.7965,Z 127,A 135.0148,B 24.9434,C -1.7386,E1 24.879,E2 311.0745} C_DIS
LIN {X -93.7862,Y 76.3535,Z 127,A 137.18,B 24.9436,C -1.7342,E1 24.8751,E2 308.9097} C_DIS
LIN {X -97.0149,Y 72.2083,Z 127,A 139.7397,B 24.9439,C -1.7305,E1 24.8707,E2 306.3467} C_DIS
LIN {X -99.7031,Y 68.4499,Z 127,A 141.9635,B 24.9442,C -1.7259,E1 24.8672,E2 304.123} C_DIS
LIN {X -101.7806,Y 65.3173,Z 127,A 143.6666,B 24.9447,C -1.7175,E1 24.8646,E2 302.4313} C_DIS
LIN {X -103.748,Y 62.1489,Z 127,A 145.4783,B 24.9449,C -1.7143,E1 24.862,E2 300.6179} C_DIS
LIN {X -106.8082,Y 56.7259,Z 127,A 148.3658,B 24.9457,C -1.7028,E1 24.8581,E2 297.7425} C_DIS
LIN {X -108.3525,Y 53.7158,Z 127,A 150.3976,B 24.9448,C -1.7166,E1 24.8555,E2 295.667} C_DIS
LIN {X -109.9183,Y 50.4385,Z 127,A 151.8609,B 24.9458,C -1.7002,E1 24.8538,E2 294.2349} C_DIS
LIN {X -111.5018,Y 46.8296,Z 127,A 153.6351,B 24.9464,C -1.6904,E1 24.8519,E2 292.474} C_DIS
LIN {X -112.4659,Y 44.4649,Z 127,A 155.4424,B 24.945,C -1.7125,E1 24.85,E2 290.6039} C_DIS
LIN {X -114.0449,Y 40.2422,Z 127,A 156.86,B 24.9474,C -1.6747,E1 24.8487,E2 289.2684} C_DIS
LIN {X -114.9616,Y 37.5443,Z 127,A 158.3935,B 24.9472,C -1.6783,E1 24.8473,E2 287.7175} C_DIS
LIN {X -116.1031,Y 33.8531,Z 127,A 160.336,B 24.9472,C -1.6773,E1 24.8458,E2 285.7663} C_DIS
LIN {X -117.2008,Y 29.8276,Z 127,A 162.2311,B 24.9479,C -1.6675,E1 24.8444,E2 283.8836} C_DIS
LIN {X -118.0727,Y 26.1657,Z 127,A 163.9889,B 24.9483,C -1.6606,E1 24.8433,E2 282.1319} C_DIS
LIN {X -118.7421,Y 22.934,Z 127,A 165.547,B 24.9487,C -1.6553,E1 24.8425,E2 280.5771} C_DIS
LIN {X -119.4,Y 19.2279,Z 127,A 167.4697,B 24.9487,C -1.6555,E1 24.8416,E2 278.6427} C_DIS
LIN {X -119.9385,Y 15.5045,Z 127,A 169.0686,B 24.9495,C -1.6418,E1 24.841,E2 277.0668} C_DIS
LIN {X -120.3361,Y 12.0488,Z 127,A 170.9056,B 24.9493,C -1.6445,E1 24.8404,E2 275.2123} C_DIS
LIN {X -120.6571,Y 8.217,Z 127,A 172.4165,B 24.9505,C -1.6253,E1 24.8401,E2 273.7383} C_DIS
LIN {X -120.8248,Y 5.1969,Z 127,A 174.0475,B 24.9503,C -1.629,E1 24.8399,E2 272.0884} C_DIS
LIN {X -120.915,Y 2.2799,Z 127,A 175.4531,B 24.9505,C -1.6255,E1 24.8398,E2 270.6828} C_DIS
LIN {X -120.9297,Y -1.4841,Z 127,A 177.3776,B 24.9505,C -1.6257,E1 24.8398,E2 268.7461} C_DIS
LIN {X -120.8433,Y -4.7664,Z 127,A 178.912,B 24.9508,C -1.6198,E1 24.84,E2 267.2168} C_DIS
LIN {X -120.6414,Y -8.4486,Z 127,A -179.3215,B 24.9511,C -1.6149,E1 24.8403,E2 265.4512} C_DIS
LIN {X -120.307,Y -12.3261,Z 127,A -177.4728,B 24.9515,C -1.6092,E1 24.8408,E2 263.6051} C_DIS
LIN {X -119.8053,Y -16.5101,Z 127,A -175.4342,B 24.9518,C -1.6046,E1 24.8415,E2 261.5652} C_DIS
LIN {X -119.152,Y -20.7106,Z 127,A -173.4043,B 24.9521,C -1.5988,E1 24.8424,E2 259.537} C_DIS
LIN {X -118.4842,Y -24.2313,Z 127,A -171.8251,B 24.9527,C -1.5884,E1 24.8433,E2 257.9734} C_DIS
LIN {X -117.8225,Y -27.2673,Z 127,A -170.3472,B 24.953,C -1.584,E1 24.8442,E2 256.4971} C_DIS
LIN {X -117.0926,Y -30.2486,Z 127,A -168.3945,B 24.952,C -1.6011,E1 24.8456,E2 254.4923} C_DIS
LIN {X -116.0605,Y -33.9968,Z 127,A -167.0351,B 24.9536,C -1.5745,E1 24.8466,E2 253.1885} C_DIS
LIN {X -115.1149,Y -37.0706,Z 127,A -165.4853,B 24.9538,C -1.571,E1 24.8479,E2 251.6382} C_DIS
LIN {X -113.3906,Y -42.0552,Z 127,A -162.8082,B 24.9538,C -1.5712,E1 24.8504,E2 248.9455} C_DIS
LIN {X -111.9878,Y -45.655,Z 127,A -161.0666,B 24.9543,C -1.5619,E1 24.8522,E2 247.2161} C_DIS
LIN {X -110.3877,Y -49.3993,Z 127,A -159.1993,B 24.9548,C -1.5536,E1 24.8543,E2 245.3583} C_DIS
LIN {X -108.9616,Y -52.4692,Z 127,A -157.5529,B 24.9549,C -1.5509,E1 24.8562,E2 243.7094} C_DIS
LIN {X -107.3165,Y -55.7607,Z 127,A -155.7368,B 24.955,C -1.5492,E1 24.8586,E2 241.8878} C_DIS
LIN {X -105.9281,Y -58.3552,Z 127,A -154.2489,B 24.955,C -1.5494,E1 24.8606,E2 240.3914} C_DIS
LIN {X -104.0929,Y -61.5656,Z 127,A -152.651,B 24.9557,C -1.538,E1 24.8628,E2 238.8125} C_DIS
LIN {X -102.7104,Y -63.8458,Z 127,A -151.2256,B 24.9555,C -1.5417,E1 24.8649,E2 237.371} C_DIS
LIN {X -100.2518,Y -67.6406,Z 127,A -149.2315,B 24.9562,C -1.5296,E1 24.8679,E2 235.3957} C_DIS
LIN {X -98.1527,Y -70.6537,Z 127,A -147.4982,B 24.9564,C -1.5249,E1 24.8707,E2 233.6651} C_DIS
LIN {X -95.6378,Y -74.021,Z 127,A -145.3804,B 24.9564,C -1.5256,E1 24.8743,E2 231.5355} C_DIS
LIN {X -93.0961,Y -77.193,Z 127,A -143.6924,B 24.9573,C -1.5105,E1 24.8772,E2 229.8757} C_DIS
LIN {X -91.2077,Y -79.4156,Z 127,A -142.1801,B 24.9571,C -1.513,E1 24.88,E2 228.3504} C_DIS
LIN {X -88.9907,Y -81.8922,Z 127,A -140.5336,B 24.9571,C -1.5126,E1 24.8831,E2 226.6975} C_DIS
LIN {X -86.2376,Y -84.7868,Z 127,A -138.6826,B 24.9575,C -1.5066,E1 24.8867,E2 224.8528} C_DIS
LIN {X -84.0549,Y -86.9509,Z 127,A -137.1558,B 24.9575,C -1.5066,E1 24.8898,E2 223.3196} C_DIS
LIN {X -81.1288,Y -89.6892,Z 127,A -135.2778,B 24.9577,C -1.5018,E1 24.8936,E2 221.4454} C_DIS
LIN {X -78.523,Y -91.9771,Z 127,A -133.6699,B 24.958,C -1.4971,E1 24.897,E2 219.8426} C_DIS
LIN {X -75.9523,Y -94.1114,Z 127,A -131.9712,B 24.9579,C -1.4992,E1 24.9007,E2 218.1322} C_DIS
LIN {X -73.1109,Y -96.3368,Z 127,A -130.1979,B 24.9579,C -1.499,E1 24.9046,E2 216.3532} C_DIS
LIN {X -69.5676,Y -98.9264,Z 127,A -128.1713,B 24.9582,C -1.493,E1 24.9092,E2 214.3337} C_DIS
LIN {X -66.4278,Y -101.0595,Z 127,A -126.1852,B 24.9579,C -1.4986,E1 24.9139,E2 212.3277} C_DIS
LIN {X -62.9728,Y -103.2478,Z 127,A -124.4915,B 24.9587,C -1.4846,E1 24.9178,E2 210.662} C_DIS
LIN {X -60.4607,Y -104.7387,Z 127,A -123.2082,B 24.9591,C -1.478,E1 24.9209,E2 209.3905} C_DIS
LIN {X -57.9254,Y -106.1621,Z 127,A -121.647,B 24.9587,C -1.4845,E1 24.9248,E2 207.8095} C_DIS
LIN {X -54.4876,Y -107.9682,Z 127,A -119.763,B 24.9587,C -1.4841,E1 24.9295,E2 205.9214} C_DIS
LIN {X -50.3099,Y -109.9774,Z 127,A -117.3799,B 24.9584,C -1.4901,E1 24.9355,E2 203.5181} C_DIS
LIN {X -46.6773,Y -111.566,Z 127,A -115.7682,B 24.9592,C -1.4758,E1 24.9396,E2 201.9364} C_DIS
LIN {X -43.0229,Y -113.0253,Z 127,A -113.9453,B 24.9594,C -1.4721,E1 24.9443,E2 200.1184} C_DIS
LIN {X -40.1153,Y -114.0895,Z 127,A -112.4784,B 24.9594,C -1.4708,E1 24.9482,E2 198.6516} C_DIS
LIN {X -36.3792,Y -115.3367,Z 127,A -110.694,B 24.9598,C -1.4656,E1 24.9529,E2 196.8765} C_DIS
LIN {X -33.1203,Y -116.313,Z 127,A -108.9391,B 24.9595,C -1.4711,E1 24.9576,E2 195.1056} C_DIS
LIN {X -29.4106,Y -117.308,Z 127,A -107.0501,B 24.9593,C -1.4732,E1 24.9628,E2 193.2089} C_DIS
LIN {X -25.6074,Y -118.1945,Z 127,A -105.2839,B 24.9596,C -1.4684,E1 24.9676,E2 191.4518} C_DIS
LIN {X -22.8756,Y -118.7533,Z 127,A -103.5855,B 24.9587,C -1.4855,E1 24.9723,E2 189.711} C_DIS
LIN {X -19.3169,Y -119.3852,Z 127,A -102.3364,B 24.9599,C -1.4633,E1 24.9756,E2 188.5133} C_DIS
LIN {X -15.0745,Y -119.9943,Z 127,A -100.1245,B 24.9594,C -1.4713,E1 24.9818,E2 186.2807} C_DIS
LIN {X -11.6931,Y -120.3713,Z 127,A -98.2499,B 24.9588,C -1.4835,E1 24.9871,E2 184.3762} C_DIS
LIN {X -8.37,Y -120.6467,Z 127,A -96.7753,B 24.959,C -1.4786,E1 24.9912,E2 182.9128} C_DIS
LIN {X -3.4152,Y -120.8887,Z 127,A -94.6463,B 24.9596,C -1.4684,E1 24.9971,E2 180.8075} C_DIS
LIN {X 0.2341,Y -120.9374,Z 127,A -92.5257,B 24.9586,C -1.4873,E1 25.0031,E2 178.6421} C_DIS
LIN {X 0.2341,Y -120.9374,Z 127,A -92.5257,B 24.9586,C -1.4873,E1 25.0031,E2 178.6421} C_DIS
Enddeposition()
LIN {X 0.8258,Y -120.0661,Z 127,A -91.9917,B 24.957,C -1.5143,E1 25.0048,E2 178.0442} C_DIS
Startdeposition()
$VEL.CP = VEL_PRINT
LIN {X -0.231,Y -120.0819,Z 127,A -94.815,B 24.963,C -1.4063,E1 24.9962,E2 181.1233} C_DIS
LIN {X -6.016,Y -119.9318,Z 127,A -97.4811,B 24.9627,C -1.4104,E1 24.9888,E2 183.7805} C_DIS
LIN {X -11.2671,Y -119.5515,Z 127,A -99.0731,B 24.9605,C -1.4524,E1 24.9846,E2 185.2736} C_DIS
LIN {X -17.6876,Y -118.7731,Z 127,A -102.5026,B 24.9613,C -1.4372,E1 24.975,E2 188.7415} C_DIS
LIN {X -21.9903,Y -118.0526,Z 127,A -104.3342,B 24.9607,C -1.4493,E1 24.97,E2 190.5464} C_DIS
LIN {X -25.3859,Y -117.3672,Z 127,A -106.0359,B 24.9607,C -1.4478,E1 24.9654,E2 192.2535} C_DIS
LIN {X -28.5496,Y -116.6378,Z 127,A -107.5692,B 24.9607,C -1.4493,E1 24.9612,E2 193.7852} C_DIS
LIN {X -32.0711,Y -115.7211,Z 127,A -109.4267,B 24.9609,C -1.4449,E1 24.9562,E2 195.656} C_DIS
LIN {X -35.5961,Y -114.6838,Z 127,A -111.4676,B 24.9615,C -1.4333,E1 24.9506,E2 197.728} C_DIS
LIN {X -39.0308,Y -113.5629,Z 127,A -112.745,B 24.9604,C -1.4547,E1 24.9474,E2 198.957} C_DIS
LIN {X -41.8486,Y -112.5552,Z 127,A -114.3078,B 24.9606,C -1.45,E1 24.9432,E2 200.5343} C_DIS
LIN {X -46.0452,Y -110.904,Z 127,A -116.354,B 24.9602,C -1.4569,E1 24.938,E2 202.5686} C_DIS
LIN {X -49.8468,Y -109.2477,Z 127,A -118.5095,B 24.9605,C -1.4512,E1 24.9324,E2 204.7428} C_DIS
LIN {X -54.4027,Y -107.0508,Z 127,A -120.7955,B 24.9601,C -1.4599,E1 24.9267,E2 207.0141} C_DIS
LIN {X -57.5854,Y -105.3732,Z 127,A -122.4482,B 24.9598,C -1.465,E1 24.9227,E2 208.6593} C_DIS
LIN {X -60.4508,Y -103.7575,Z 127,A -124.184,B 24.9601,C -1.4598,E1 24.9184,E2 210.4124} C_DIS
LIN {X -63.5952,Y -101.8583,Z 127,A -125.9805,B 24.9601,C -1.4606,E1 24.9142,E2 212.2128} C_DIS
LIN {X -67.2081,Y -99.5115,Z 127,A -127.9546,B 24.9597,C -1.4675,E1 24.9096,E2 214.1769} C_DIS
LIN {X -71.669,Y -96.3501,Z 127,A -130.6345,B 24.9596,C -1.4689,E1 24.9035,E2 216.8629} C_DIS
LIN {X -74.6293,Y -94.0743,Z 127,A -132.3825,B 24.9593,C -1.4736,E1 24.8997,E2 218.6061} C_DIS
LIN {X -78.7484,Y -90.6545,Z 127,A -134.9201,B 24.959,C -1.4793,E1 24.8943,E2 221.14} C_DIS
LIN {X -81.3815,Y -88.2982,Z 127,A -136.7118,B 24.959,C -1.4781,E1 24.8905,E2 222.9417} C_DIS
LIN {X -84.497,Y -85.3214,Z 127,A -138.6333,B 24.9585,C -1.4883,E1 24.8867,E2 224.8469} C_DIS
LIN {X -86.8224,Y -82.9554,Z 127,A -140.4486,B 24.9589,C -1.4817,E1 24.8831,E2 226.6858} C_DIS
LIN {X -90.0299,Y -79.4636,Z 127,A -142.6825,B 24.9585,C -1.4881,E1 24.879,E2 228.9144} C_DIS
LIN {X -92.3799,Y -76.7165,Z 127,A -144.2458,B 24.9579,C -1.4991,E1 24.8762,E2 230.4586} C_DIS
LIN {X -94.7729,Y -73.7419,Z 127,A -146.602,B 24.9589,C -1.4806,E1 24.8721,E2 232.87} C_DIS
LIN {X -97.2578,Y -70.4327,Z 127,A -147.972,B 24.9572,C -1.5114,E1 24.8699,E2 234.1732} C_DIS
LIN {X -101.7306,Y -63.7996,Z 127,A -151.626,B 24.9562,C -1.5283,E1 24.8643,E2 237.8052} C_DIS
LIN {X -103.2261,Y -61.3507,Z 127,A -153.3095,B 24.9568,C -1.5185,E1 24.8618,E2 239.5208} C_DIS
LIN {X -105.8836,Y -56.6445,Z 127,A -155.9576,B 24.9566,C -1.5226,E1 24.8582,E2 242.173} C_DIS
LIN {X -107.6153,Y -53.2766,Z 127,A -157.7486,B 24.9562,C -1.5284,E1 24.8559,E2 243.9599} C_DIS
LIN {X -110.0112,Y -48.1355,Z 127,A -160.1164,B 24.955,C -1.5506,E1 24.8532,E2 246.2877} C_DIS
LIN {X -111.188,Y -45.3508,Z 127,A -161.8626,B 24.9555,C -1.5419,E1 24.8513,E2 248.0644} C_DIS
LIN {X -112.4338,Y -42.1693,Z 127,A -163.955,B 24.9563,C -1.5272,E1 24.8492,E2 250.2036} C_DIS
LIN {X -113.695,Y -38.6393,Z 127,A -165.0637,B 24.9543,C -1.5613,E1 24.8483,E2 251.2372} C_DIS
LIN {X -114.4166,Y -36.4499,Z 127,A -167.3031,B 24.9569,C -1.5168,E1 24.8463,E2 253.5957} C_DIS
LIN {X -116.0363,Y -30.9065,Z 127,A -169.4945,B 24.9551,C -1.5488,E1 24.8447,E2 255.7234} C_DIS
LIN {X -117.2702,Y -25.8303,Z 127,A -171.7087,B 24.9539,C -1.5683,E1 24.8433,E2 257.9041} C_DIS
LIN {X -118.0304,Y -22.1052,Z 127,A -174.0365,B 24.9548,C -1.5525,E1 24.8421,E2 260.2834} C_DIS
LIN {X -118.6957,Y -18.1883,Z 127,A -175.427,B 24.9532,C -1.5797,E1 24.8415,E2 261.6173} C_DIS
LIN {X -119.217,Y -14.3855,Z 127,A -177.349,B 24.9532,C -1.5818,E1 24.8408,E2 263.5459} C_DIS
LIN {X -119.5858,Y -10.8955,Z 127,A -178.988,B 24.9527,C -1.5887,E1 24.8403,E2 265.1782} C_DIS
LIN {X -119.8866,Y -6.8341,Z 127,A 179.0936,B 24.9523,C -1.596,E1 24.84,E2 267.0906} C_DIS
LIN {X -120.0337,Y -3.3843,Z 127,A 177.4713,B 24.9519,C -1.6024,E1 24.8398,E2 268.7075} C_DIS
LIN {X -120.0826,Y -0.1696,Z 127,A 175.7427,B 24.9521,C -1.5993,E1 24.8398,E2 270.454} C_DIS
LIN {X -120.0218,Y 3.7735,Z 127,A 173.9369,B 24.9515,C -1.6086,E1 24.8399,E2 272.2485} C_DIS
LIN {X -119.8206,Y 7.907,Z 127,A 171.9721,B 24.9511,C -1.6155,E1 24.8402,E2 274.2087} C_DIS
LIN {X -119.5378,Y 11.415,Z 127,A 170.3496,B 24.9506,C -1.6233,E1 24.8406,E2 275.8222} C_DIS
LIN {X -119.1862,Y 14.6485,Z 127,A 168.6571,B 24.9506,C -1.6225,E1 24.8412,E2 277.5268} C_DIS
LIN {X -118.6681,Y 18.367,Z 127,A 166.9367,B 24.9501,C -1.6313,E1 24.8418,E2 279.2364} C_DIS
LIN {X -118.1,Y 21.7273,Z 127,A 165.2292,B 24.9501,C -1.6332,E1 24.8427,E2 280.9496} C_DIS
LIN {X -117.3104,Y 25.6461,Z 127,A 163.345,B 24.9496,C -1.6404,E1 24.8438,E2 282.8279} C_DIS
LIN {X -116.4637,Y 29.2589,Z 127,A 161.5636,B 24.9493,C -1.6456,E1 24.8449,E2 284.6072} C_DIS
LIN {X -115.0242,Y 34.482,Z 127,A 159.0247,B 24.9486,C -1.6558,E1 24.8469,E2 287.1365} C_DIS
LIN {X -113.2838,Y 39.8276,Z 127,A 155.762,B 24.9496,C -1.64,E1 24.8498,E2 290.4553} C_DIS
LIN {X -111.8451,Y 43.7054,Z 127,A 154.5787,B 24.9472,C -1.6793,E1 24.8509,E2 291.5518} C_DIS
LIN {X -110.8567,Y 46.1574,Z 127,A 152.9539,B 24.9479,C -1.6679,E1 24.8527,E2 293.2128} C_DIS
LIN {X -109.3767,Y 49.5606,Z 127,A 150.8872,B 24.9483,C -1.6609,E1 24.8551,E2 295.3074} C_DIS
LIN {X -107.9066,Y 52.6875,Z 127,A 149.6764,B 24.9468,C -1.6842,E1 24.8565,E2 296.4693} C_DIS
LIN {X -106.3386,Y 55.7817,Z 127,A 147.2681,B 24.9485,C -1.6577,E1 24.8597,E2 298.9536} C_DIS
LIN {X -104.0655,Y 59.9153,Z 127,A 145.5225,B 24.9468,C -1.6854,E1 24.862,E2 300.6423} C_DIS
LIN {X -101.8706,Y 63.5754,Z 127,A 143.5909,B 24.9461,C -1.6957,E1 24.8648,E2 302.5593} C_DIS
LIN {X -99.8678,Y 66.681,Z 127,A 141.509,B 24.9467,C -1.6872,E1 24.868,E2 304.6718} C_DIS
LIN {X -96.7326,Y 71.15,Z 127,A 138.7554,B 24.9466,C -1.6882,E1 24.8726,E2 307.4365} C_DIS
LIN {X -94.4135,Y 74.2001,Z 127,A 137.6028,B 24.9444,C -1.7217,E1 24.8744,E2 308.5148} C_DIS
LIN {X -91.0372,Y 78.3072,Z 127,A 134.8822,B 24.9445,C -1.7205,E1 24.8793,E2 311.2507} C_DIS
LIN {X -88.9757,Y 80.6431,Z 127,A 133.0078,B 24.9453,C -1.7079,E1 24.8829,E2 313.1636} C_DIS
LIN {X -85.2204,Y 84.5992,Z 127,A 130.441,B 24.9448,C -1.7159,E1 24.8878,E2 315.7224} C_DIS
LIN {X -82.1552,Y 87.5785,Z 127,A 128.6781,B 24.9437,C -1.7325,E1 24.8913,E2 317.4529} C_DIS
LIN {X -79.7358,Y 89.788,Z 127,A 126.9063,B 24.9441,C -1.7273,E1 24.8951,E2 319.2443} C_DIS
LIN {X -77.1947,Y 91.9824,Z 127,A 125.3734,B 24.9437,C -1.7338,E1 24.8983,E2 320.7675} C_DIS
LIN {X -72.7015,Y 95.5744,Z 127,A 122.7794,B 24.9429,C -1.7462,E1 24.904,E2 323.3416} C_DIS
LIN {X -67.4572,Y 99.3429,Z 127,A 119.9281,B 24.9418,C -1.7625,E1 24.9104,E2 326.1641} C_DIS
LIN {X -63.7911,Y 101.7359,Z 127,A 116.6241,B 24.9449,C -1.7144,E1 24.9185,E2 329.5931} C_DIS
LIN {X -58.7252,Y 104.7418,Z 127,A 114.6931,B 24.9421,C -1.7571,E1 24.9229,E2 331.4282} C_DIS
LIN {X -55.5565,Y 106.4572,Z 127,A 112.9482,B 24.9421,C -1.7589,E1 24.9272,E2 333.1737} C_DIS
LIN {X -51.5323,Y 108.4627,Z 127,A 110.5895,B 24.9424,C -1.7531,E1 24.9332,E2 335.5523} C_DIS
LIN {X -48.2282,Y 109.9707,Z 127,A 109.0904,B 24.9416,C -1.7658,E1 24.9369,E2 337.0247} C_DIS
LIN {X -45.2147,Y 111.2434,Z 127,A 106.9428,B 24.9431,C -1.7426,E1 24.9426,E2 339.2323} C_DIS
LIN {X -41.1078,Y 112.8255,Z 127,A 105.3998,B 24.9413,C -1.7696,E1 24.9465,E2 340.7144} C_DIS
LIN {X -37.3448,Y 114.127,Z 127,A 103.4747,B 24.9413,C -1.7708,E1 24.9516,E2 342.6402} C_DIS
LIN {X -34.1107,Y 115.1343,Z 127,A 101.8231,B 24.9413,C -1.7711,E1 24.956,E2 344.294} C_DIS
LIN {X -28.7257,Y 116.5949,Z 127,A 99.2008,B 24.9409,C -1.7755,E1 24.9631,E2 346.9095} C_DIS
LIN {X -25.6284,Y 117.3143,Z 127,A 97.7218,B 24.9407,C -1.7786,E1 24.9671,E2 348.3831} C_DIS
LIN {X -22.1674,Y 118.0185,Z 127,A 95.9582,B 24.9408,C -1.7765,E1 24.972,E2 350.1537} C_DIS
LIN {X -17.947,Y 118.733,Z 127,A 94.0504,B 24.9404,C -1.7839,E1 24.9772,E2 352.0456} C_DIS
LIN {X -15.1037,Y 119.1278,Z 127,A 91.9329,B 24.9425,C -1.7517,E1 24.9833,E2 354.2412} C_DIS
LIN {X -10.2582,Y 119.644,Z 127,A 90.3466,B 24.9402,C -1.7856,E1 24.9875,E2 355.7479} C_DIS
LIN {X -4.7153,Y 119.9892,Z 127,A 87.712,B 24.9402,C -1.7872,E1 24.9948,E2 358.3793} C_DIS
LIN {X -2.0256,Y 120.0641,Z 127,A 85.7494,B 24.9421,C -1.7572,E1 25.0005,E2 360.4132} C_DIS
LIN {X 2.4017,Y 120.0572,Z 127,A 84.2899,B 24.9402,C -1.7868,E1 25.0044,E2 361.8024} C_DIS
LIN {X 6.9824,Y 119.8784,Z 127,A 82.1447,B 24.94,C -1.7888,E1 25.0103,E2 363.9422} C_DIS
LIN {X 9.6697,Y 119.6911,Z 127,A 80.6906,B 24.9405,C -1.7811,E1 25.0144,E2 365.4139} C_DIS
LIN {X 14.2264,Y 119.2356,Z 127,A 78.7091,B 24.9399,C -1.79,E1 25.0198,E2 367.373} C_DIS
LIN {X 16.8864,Y 118.8878,Z 127,A 77.3078,B 24.9403,C -1.7842,E1 25.0238,E2 368.7869} C_DIS
LIN {X 19.9319,Y 118.4153,Z 127,A 75.8537,B 24.9403,C -1.7844,E1 25.0278,E2 370.239} C_DIS
LIN {X 22.9122,Y 117.8751,Z 127,A 74.4049,B 24.9403,C -1.7837,E1 25.0317,E2 371.6878} C_DIS
LIN {X 26.3104,Y 117.1655,Z 127,A 72.5973,B 24.9409,C -1.7759,E1 25.0367,E2 373.5116} C_DIS
LIN {X 29.8818,Y 116.3036,Z 127,A 71.0195,B 24.9404,C -1.7829,E1 25.0409,E2 375.0703} C_DIS
LIN {X 32.7885,Y 115.5178,Z 127,A 69.1743,B 24.9417,C -1.7632,E1 25.046,E2 376.9593} C_DIS
LIN {X 36.1097,Y 114.5245,Z 127,A 67.9512,B 24.9405,C -1.7816,E1 25.0492,E2 378.1364} C_DIS
LIN {X 38.9009,Y 113.6068,Z 127,A 66.4317,B 24.9409,C -1.775,E1 25.0532,E2 379.6687} C_DIS
LIN {X 42.826,Y 112.1851,Z 127,A 64.5306,B 24.9408,C -1.7774,E1 25.0582,E2 381.5603} C_DIS
LIN {X 46.7172,Y 110.6208,Z 127,A 62.4699,B 24.9411,C -1.7725,E1 25.0635,E2 383.6277} C_DIS
LIN {X 50.438,Y 108.9749,Z 127,A 60.5735,B 24.9411,C -1.7723,E1 25.0683,E2 385.5198} C_DIS
LIN {X 53.3671,Y 107.5705,Z 127,A 59.0812,B 24.9411,C -1.7731,E1 25.0721,E2 387.0063} C_DIS
LIN {X 56.0926,Y 106.1748,Z 127,A 57.5667,B 24.9414,C -1.7686,E1 25.0758,E2 388.5271} C_DIS
LIN {X 60.2773,Y 103.8575,Z 127,A 54.8436,B 24.9429,C -1.7448,E1 25.0826,E2 391.2985} C_DIS
LIN {X 63.4392,Y 101.9557,Z 127,A 53.8027,B 24.9409,C -1.7758,E1 25.0849,E2 392.2629} C_DIS
LIN {X 67.9744,Y 98.9917,Z 127,A 51.0312,B 24.9418,C -1.7627,E1 25.0914,E2 395.056} C_DIS
LIN {X 70.5881,Y 97.144,Z 127,A 49.3421,B 24.9424,C -1.7524,E1 25.0952,E2 396.7635} C_DIS
LIN {X 73.3709,Y 95.0588,Z 127,A 47.7747,B 24.9424,C -1.7538,E1 25.0987,E2 398.322} C_DIS
LIN {X 76.1538,Y 92.8469,Z 127,A 46.1424,B 24.9424,C -1.7536,E1 25.1022,E2 399.9488} C_DIS
LIN {X 78.5535,Y 90.8248,Z 127,A 44.4792,B 24.9431,C -1.7427,E1 25.1058,E2 401.631} C_DIS
LIN {X 81.5574,Y 88.1368,Z 127,A 42.7441,B 24.9428,C -1.7478,E1 25.1094,E2 403.3473} C_DIS
LIN {X 84.0793,Y 85.7339,Z 127,A 40.9219,B 24.9435,C -1.7366,E1 25.1131,E2 405.1883} C_DIS
LIN {X 86.7453,Y 83.0354,Z 127,A 39.198,B 24.9435,C -1.7367,E1 25.1164,E2 406.9044} C_DIS
LIN {X 89.5618,Y 79.9885,Z 127,A 37.2832,B 24.9435,C -1.7353,E1 25.12,E2 408.8141} C_DIS
LIN {X 91.8428,Y 77.3616,Z 127,A 35.281,B 24.9449,C -1.715,E1 25.1237,E2 410.8551} C_DIS
LIN {X 95.2845,Y 73.0779,Z 127,A 33.0176,B 24.9442,C -1.7258,E1 25.1275,E2 413.0823} C_DIS
LIN {X 97.3327,Y 70.33,Z 127,A 31.2376,B 24.9449,C -1.7147,E1 25.1305,E2 414.88} C_DIS
LIN {X 99.6225,Y 67.0442,Z 127,A 29.5211,B 24.9446,C -1.7192,E1 25.1332,E2 416.5775} C_DIS
LIN {X 101.6291,Y 63.962,Z 127,A 27.3843,B 24.9461,C -1.6961,E1 25.1365,E2 418.7579} C_DIS
LIN {X 103.318,Y 61.1952,Z 127,A 25.6391,B 24.947,C -1.6824,E1 25.139,E2 420.5265} C_DIS
LIN {X 105.4285,Y 57.4835,Z 127,A 24.4133,B 24.9448,C -1.716,E1 25.1405,E2 421.6668} C_DIS
LIN {X 107.5138,Y 53.4814,Z 127,A 22.0092,B 24.946,C -1.6977,E1 25.1436,E2 424.1012} C_DIS
LIN {X 108.9533,Y 50.4843,Z 127,A 20.4888,B 24.946,C -1.6964,E1 25.1454,E2 425.6166} C_DIS
LIN {X 110.267,Y 47.5486,Z 127,A 18.7907,B 24.9469,C -1.684,E1 25.1474,E2 427.3347} C_DIS
LIN {X 111.7002,Y 44.0744,Z 127,A 16.7064,B 24.9481,C -1.6646,E1 25.1496,E2 429.4532} C_DIS
LIN {X 113.0508,Y 40.4901,Z 127,A 15.396,B 24.9468,C -1.6842,E1 25.1508,E2 430.7101} C_DIS
LIN {X 114.3214,Y 36.7441,Z 127,A 13.4571,B 24.9474,C -1.6759,E1 25.1525,E2 432.6573} C_DIS
LIN {X 115.6036,Y 32.486,Z 127,A 11.4005,B 24.9476,C -1.6726,E1 25.1541,E2 434.7101} C_DIS
LIN {X 116.3562,Y 29.6772,Z 127,A 9.9801,B 24.9479,C -1.6667,E1 25.1551,E2 436.1363} C_DIS
LIN {X 117.2217,Y 26.0528,Z 127,A 8.1369,B 24.9485,C -1.6579,E1 25.1563,E2 437.9895} C_DIS
LIN {X 117.9882,Y 22.3243,Z 127,A 6.2709,B 24.949,C -1.6497,E1 25.1573,E2 439.8639} C_DIS
LIN {X 118.6718,Y 18.3425,Z 127,A 4.4429,B 24.949,C -1.6484,E1 25.1581,E2 441.6842} C_DIS
LIN {X 119.3233,Y 13.4766,Z 127,A 2.196,B 24.9493,C -1.6456,E1 25.1589,E2 443.9246} C_DIS
LIN {X 119.6502,Y 10.1814,Z 127,A -0.1283,B 24.9518,C -1.6041,E1 25.1595,E2 446.3328} C_DIS
LIN {X 119.9658,Y 5.2609,Z 127,A -2.4326,B 24.9521,C -1.5988,E1 25.1597,E2 448.6358} C_DIS
LIN {X 120.0815,Y 0.3614,Z 127,A -4.0873,B 24.9505,C -1.6245,E1 25.1597,E2 450.2202} C_DIS
LIN {X 119.8793,Y -6.9661,Z 127,A -7.1195,B 24.9498,C -1.636,E1 25.1596,E2 453.2073} C_DIS
LIN {X 119.411,Y -12.6686,Z 127,A -10.2826,B 24.9517,C -1.6056,E1 25.1588,E2 456.4232} C_DIS
LIN {X 118.7894,Y -17.5641,Z 127,A -12.9063,B 24.9529,C -1.5847,E1 25.1578,E2 459.0807} C_DIS
LIN {X 118.2789,Y -20.7321,Z 127,A -14.2335,B 24.9527,C -1.5897,E1 25.1571,E2 460.3885} C_DIS
LIN {X 117.6321,Y -24.1275,Z 127,A -15.7433,B 24.9526,C -1.5912,E1 25.1563,E2 461.8859} C_DIS
LIN {X 116.4722,Y -29.2256,Z 127,A -18.3482,B 24.9534,C -1.5777,E1 25.1547,E2 464.5076} C_DIS
LIN {X 115.5434,Y -32.6983,Z 127,A -19.9703,B 24.9534,C -1.5767,E1 25.1535,E2 466.1225} C_DIS
LIN {X 114.6333,Y -35.7588,Z 127,A -21.4605,B 24.9536,C -1.5735,E1 25.1522,E2 467.6118} C_DIS
LIN {X 113.4188,Y -39.4428,Z 127,A -23.3303,B 24.954,C -1.5667,E1 25.1506,E2 469.4871} C_DIS
LIN {X 112.1301,Y -42.971,Z 127,A -25.0888,B 24.9542,C -1.5627,E1 25.1488,E2 471.2452} C_DIS
LIN {X 109.9626,Y -48.2469,Z 127,A -27.8484,B 24.9548,C -1.5524,E1 25.1459,E2 474.0139} C_DIS
LIN {X 107.9021,Y -52.6978,Z 127,A -30.1712,B 24.9552,C -1.5461,E1 25.1431,E2 476.3391} C_DIS
LIN {X 106.253,Y -55.9442,Z 127,A -31.8454,B 24.9553,C -1.544,E1 25.1409,E2 478.0094} C_DIS
LIN {X 103.6787,Y -60.585,Z 127,A -35.1246,B 24.9578,C -1.5002,E1 25.1363,E2 481.3749} C_DIS
LIN {X 100.9141,Y -65.0836,Z 127,A -36.8481,B 24.9561,C -1.5316,E1 25.1338,E2 483.0157} C_DIS
LIN {X 98.4621,Y -68.7367,Z 127,A -39.0041,B 24.9566,C -1.5229,E1 25.1304,E2 485.1817} C_DIS
LIN {X 94.2151,Y -74.4511,Z 127,A -41.9551,B 24.9558,C -1.5353,E1 25.1256,E2 488.0892} C_DIS
LIN {X 89.2787,Y -80.3047,Z 127,A -46.8513,B 24.9598,C -1.4655,E1 25.1163,E2 493.1279} C_DIS
LIN {X 85.2153,Y -84.6044,Z 127,A -48.2629,B 24.9563,C -1.5266,E1 25.1139,E2 494.3891} C_DIS
LIN {X 80.5593,Y -89.0508,Z 127,A -52.6009,B 24.9602,C -1.458,E1 25.1048,E2 498.8714} C_DIS
LIN {X 76.5361,Y -92.5298,Z 127,A -54.4129,B 24.9586,C -1.487,E1 25.101,E2 500.6079} C_DIS
LIN {X 71.4706,Y -96.4979,Z 127,A -57.7851,B 24.9597,C -1.4658,E1 25.0935,E2 504.0179} C_DIS
LIN {X 68.7026,Y -98.4858,Z 127,A -58.7346,B 24.9581,C -1.495,E1 25.0915,E2 504.8952} C_DIS
LIN {X 65.4385,Y -100.6863,Z 127,A -61.4404,B 24.9605,C -1.4515,E1 25.085,E2 507.6946} C_DIS
LIN {X 61.8014,Y -102.9586,Z 127,A -62.8377,B 24.959,C -1.4786,E1 25.0818,E2 509.0236} C_DIS
LIN {X 55.4483,Y -106.5142,Z 127,A -66.2525,B 24.9592,C -1.4752,E1 25.0735,E2 512.4364} C_DIS
LIN {X 51.9683,Y -108.2532,Z 127,A -68.2241,B 24.9597,C -1.4666,E1 25.0685,E2 514.423} C_DIS
LIN {X 48.4674,Y -109.8665,Z 127,A -70.1929,B 24.9602,C -1.4576,E1 25.0634,E2 516.4083} C_DIS
LIN {X 44.8473,Y -111.3929,Z 127,A -71.9318,B 24.96,C -1.4613,E1 25.059,E2 518.1344} C_DIS
LIN {X 40.0444,Y -113.2067,Z 127,A -75.1492,B 24.9621,C -1.422,E1 25.0503,E2 521.4381} C_DIS
LIN {X 34.9073,Y -114.8974,Z 127,A -76.8972,B 24.9602,C -1.4578,E1 25.0459,E2 523.0982} C_DIS
LIN {X 31.6272,Y -115.8416,Z 127,A -78.6277,B 24.9605,C -1.4513,E1 25.0412,E2 524.8413} C_DIS
LIN {X 28.1805,Y -116.7279,Z 127,A -80.2282,B 24.9604,C -1.4541,E1 25.0369,E2 526.4327} C_DIS
LIN {X 25.3859,Y -117.3672,Z 127,A -81.597,B 24.9604,C -1.4528,E1 25.0331,E2 527.8028} C_DIS
LIN {X 21.795,Y -118.0878,Z 127,A -84.7114,B 24.9639,C -1.3882,E1 25.0242,E2 531.0667} C_DIS
LIN {X 14.0317,Y -119.2584,Z 127,A -86.9289,B 24.9603,C -1.4562,E1 25.0185,E2 533.1214} C_DIS
LIN {X 6.3824,Y -119.9115,Z 127,A -91.726,B 24.9632,C -1.4022,E1 25.0048,E2 538.0442} C_DIS
LIN {X 0.8258,Y -120.0661,Z 127,A -91.9874,B 24.9571,C -1.5125,E1 25.0049,E2 538.0441} C_DIS
Enddeposition()
LIN {X 0.8258,Y -120.0661,Z 127,A -91.9874,B 24.9571,C -1.5125,E1 25.0049,E2 538.0441} C_DIS
Startdeposition()
$VEL.CP = VEL_PRINT
LIN {X 1.911,Y -119.2106,Z 127,A -91.5663,B 24.9566,C -1.5222,E1 25.0061,E2 537.6001} C_DIS
LIN {X 6.5482,Y -119.0456,Z 127,A -90.3315,B 24.9592,C -1.4766,E1 25.0092,E2 536.4738} C_DIS
LIN {X 12.1534,Y -118.6048,Z 127,A -87.4871,B 24.9587,C -1.4844,E1 25.0171,E2 533.6124} C_DIS
LIN {X 15.1712,Y -118.2564,Z 127,A -84.7947,B 24.9554,C -1.5436,E1 25.025,E2 530.782} C_DIS
LIN {X 21.5719,Y -117.2587,Z 127,A -82.7882,B 24.9582,C -1.4935,E1 25.0302,E2 528.8963} C_DIS
LIN {X 24.2601,Y -116.7316,Z 127,A -81.4076,B 24.958,C -1.4976,E1 25.0339,E2 527.5075} C_DIS
LIN {X 27.4427,Y -116.0259,Z 127,A -79.8669,B 24.958,C -1.4979,E1 25.0381,E2 525.9684} C_DIS
LIN {X 30.899,Y -115.1522,Z 127,A -78.0937,B 24.9577,C -1.5026,E1 25.0429,E2 524.1868} C_DIS
LIN {X 34.5362,Y -114.1158,Z 127,A -75.2838,B 24.9549,C -1.5522,E1 25.0508,E2 521.2645} C_DIS
LIN {X 40.6149,Y -112.0947,Z 127,A -73.2705,B 24.9576,C -1.505,E1 25.0558,E2 519.3669} C_DIS
LIN {X 43.6894,Y -110.9323,Z 127,A -71.6771,B 24.9574,C -1.5079,E1 25.0599,E2 517.7701} C_DIS
LIN {X 46.9131,Y -109.6099,Z 127,A -69.9948,B 24.9572,C -1.5107,E1 25.0642,E2 516.0851} C_DIS
LIN {X 50.5333,Y -107.9869,Z 127,A -68.1759,B 24.9573,C -1.5095,E1 25.0689,E2 514.2735} C_DIS
LIN {X 53.1936,Y -106.7017,Z 127,A -66.6976,B 24.957,C -1.5147,E1 25.0726,E2 512.7871} C_DIS
LIN {X 59.4841,Y -103.3266,Z 127,A -63.3727,B 24.957,C -1.5156,E1 25.0807,E2 509.4696} C_DIS
LIN {X 64.4101,Y -100.3298,Z 127,A -60.8743,B 24.9574,C -1.5077,E1 25.0866,E2 506.9975} C_DIS
LIN {X 66.612,Y -98.882,Z 127,A -59.1417,B 24.956,C -1.5327,E1 25.0908,E2 505.2117} C_DIS
LIN {X 70.7679,Y -95.9521,Z 127,A -56.5239,B 24.9552,C -1.5463,E1 25.0967,E2 502.5711} C_DIS
LIN {X 75.4163,Y -92.3434,Z 127,A -53.8958,B 24.9554,C -1.5428,E1 25.1024,E2 499.961} C_DIS
LIN {X 80.1377,Y -88.2784,Z 127,A -50.4236,B 24.9536,C -1.5732,E1 25.1098,E2 496.4309} C_DIS
LIN {X 83.3645,Y -85.2376,Z 127,A -49.0057,B 24.9554,C -1.5435,E1 25.1125,E2 495.089} C_DIS
LIN {X 85.4772,Y -83.1183,Z 127,A -46.803,B 24.953,C -1.5846,E1 25.117,E2 492.7988} C_DIS
LIN {X 88.7012,Y -79.6672,Z 127,A -44.7874,B 24.9533,C -1.5779,E1 25.1207,E2 490.8079} C_DIS
LIN {X 91.1605,Y -76.8433,Z 127,A -43.4711,B 24.9545,C -1.5589,E1 25.123,E2 489.5424} C_DIS
LIN {X 93.3291,Y -74.1925,Z 127,A -41.7409,B 24.954,C -1.5675,E1 25.126,E2 487.8} C_DIS
LIN {X 96.4821,Y -70.0441,Z 127,A -39.3125,B 24.9538,C -1.5707,E1 25.1301,E2 485.3758} C_DIS
LIN {X 99.1766,Y -66.1752,Z 127,A -36.925,B 24.953,C -1.583,E1 25.1339,E2 482.9708} C_DIS
LIN {X 102.4234,Y -61.0276,Z 127,A -34.3171,B 24.9535,C -1.5759,E1 25.1377,E2 480.3929} C_DIS
LIN {X 103.882,Y -58.5103,Z 127,A -32.5847,B 24.9522,C -1.5965,E1 25.1401,E2 478.621} C_DIS
LIN {X 105.673,Y -55.2096,Z 127,A -30.8793,B 24.9522,C -1.597,E1 25.1423,E2 476.9234} C_DIS
LIN {X 108.2773,Y -49.9096,Z 127,A -28.2619,B 24.9523,C -1.5948,E1 25.1455,E2 474.3254} C_DIS
LIN {X 110.4205,Y -44.9671,Z 127,A -25.9151,B 24.9526,C -1.5908,E1 25.1481,E2 472.0006} C_DIS
LIN {X 111.8876,Y -41.1828,Z 127,A -23.4829,B 24.9508,C -1.6207,E1 25.1505,E2 469.5116} C_DIS
LIN {X 113.4068,Y -36.7917,Z 127,A -21.4184,B 24.9508,C -1.6194,E1 25.1524,E2 467.4618} C_DIS
LIN {X 114.2901,Y -33.9486,Z 127,A -19.9996,B 24.9506,C -1.6234,E1 25.1535,E2 466.0417} C_DIS
LIN {X 115.2489,Y -30.5408,Z 127,A -17.5119,B 24.9479,C -1.668,E1 25.1554,E2 463.4632} C_DIS
LIN {X 116.4831,Y -25.4249,Z 127,A -15.8755,B 24.9501,C -1.6318,E1 25.1563,E2 461.9217} C_DIS
LIN {X 117.17,Y -22.0495,Z 127,A -13.2147,B 24.9467,C -1.6872,E1 25.1578,E2 459.1458} C_DIS
LIN {X 118.1323,Y -16.1207,Z 127,A -11.3403,B 24.9492,C -1.6461,E1 25.1585,E2 457.3792} C_DIS
LIN {X 118.4728,Y -13.3855,Z 127,A -9.9875,B 24.9489,C -1.6519,E1 25.1589,E2 456.0208} C_DIS
LIN {X 118.9779,Y -7.6879,Z 127,A -7.3554,B 24.9487,C -1.6551,E1 25.1595,E2 453.3967} C_DIS
LIN {X 119.1953,Y -2.7406,Z 127,A -4.9901,B 24.9482,C -1.6621,E1 25.1598,E2 451.0289} C_DIS
LIN {X 119.2115,Y 1.8577,Z 127,A -2.2637,B 24.9462,C -1.695,E1 25.1598,E2 448.2414} C_DIS
LIN {X 119.1029,Y 5.4146,Z 127,A -0.589,B 24.9459,C -1.6988,E1 25.1595,E2 446.5676} C_DIS
LIN {X 118.8919,Y 8.9316,Z 127,A 0.5948,B 24.9472,C -1.679,E1 25.1593,E2 445.4374} C_DIS
LIN {X 118.5378,Y 12.7929,Z 127,A 2.8773,B 24.9455,C -1.7058,E1 25.1586,E2 443.1053} C_DIS
LIN {X 118.1451,Y 16.0307,Z 127,A 4.2578,B 24.9457,C -1.7015,E1 25.1581,E2 441.743} C_DIS
LIN {X 117.5737,Y 19.7777,Z 127,A 5.8956,B 24.9459,C -1.6983,E1 25.1574,E2 440.1223} C_DIS
LIN {X 117.0141,Y 22.8588,Z 127,A 7.5158,B 24.9453,C -1.7088,E1 25.1565,E2 438.487} C_DIS
LIN {X 116.1774,Y 26.7869,Z 127,A 9.361,B 24.9452,C -1.7107,E1 25.1554,E2 436.648} C_DIS
LIN {X 115.3787,Y 30.0439,Z 127,A 10.9179,B 24.945,C -1.713,E1 25.1544,E2 435.0946} C_DIS
LIN {X 114.5415,Y 33.0963,Z 127,A 12.845,B 24.9434,C -1.7377,E1 25.1529,E2 433.1203} C_DIS
LIN {X 113.5402,Y 36.3796,Z 127,A 14.0465,B 24.9445,C -1.7207,E1 25.1519,E2 431.9658} C_DIS
LIN {X 112.5134,Y 39.4395,Z 127,A 15.8588,B 24.9434,C -1.7382,E1 25.1502,E2 430.1224} C_DIS
LIN {X 110.5917,Y 44.5464,Z 127,A 18.3074,B 24.9434,C -1.7375,E1 25.1477,E2 427.6891} C_DIS
LIN {X 109.4291,Y 47.3298,Z 127,A 19.7069,B 24.9434,C -1.7393,E1 25.1462,E2 426.2931} C_DIS
LIN {X 108.0966,Y 50.2977,Z 127,A 21.1737,B 24.9434,C -1.7391,E1 25.1445,E2 424.8347} C_DIS
LIN {X 106.6829,Y 53.2314,Z 127,A 22.867,B 24.9426,C -1.7498,E1 25.1424,E2 423.1252} C_DIS
LIN {X 104.9114,Y 56.6425,Z 127,A 25.025,B 24.9413,C -1.7701,E1 25.1395,E2 420.9306} C_DIS
LIN {X 103.1649,Y 59.7654,Z 127,A 26.2647,B 24.9425,C -1.7514,E1 25.1379,E2 419.7415} C_DIS
LIN {X 100.9942,Y 63.3636,Z 127,A 28.3491,B 24.9419,C -1.76,E1 25.1348,E2 417.6474} C_DIS
LIN {X 99.1978,Y 66.1431,Z 127,A 29.8738,B 24.9419,C -1.7609,E1 25.1325,E2 416.1281} C_DIS
LIN {X 97.1978,Y 69.0462,Z 127,A 31.5754,B 24.9416,C -1.7656,E1 25.1298,E2 414.4237} C_DIS
LIN {X 95.2407,Y 71.7213,Z 127,A 33.1911,B 24.9412,C -1.7707,E1 25.1271,E2 412.8037} C_DIS
LIN {X 91.3974,Y 76.5602,Z 127,A 36.1334,B 24.9408,C -1.7765,E1 25.1219,E2 409.8615} C_DIS
LIN {X 89.0177,Y 79.3136,Z 127,A 37.9253,B 24.9404,C -1.7827,E1 25.1186,E2 408.063} C_DIS
LIN {X 86.8316,Y 81.7007,Z 127,A 39.4246,B 24.9404,C -1.7835,E1 25.1157,E2 406.5685} C_DIS
LIN {X 84.1195,Y 84.4918,Z 127,A 41.1367,B 24.9406,C -1.78,E1 25.1124,E2 404.8719} C_DIS
LIN {X 81.4062,Y 87.1086,Z 127,A 43.1892,B 24.9396,C -1.7953,E1 25.1082,E2 402.7916} C_DIS
LIN {X 78.0457,Y 90.1325,Z 127,A 45.3806,B 24.9392,C -1.8006,E1 25.1036,E2 400.5965} C_DIS
LIN {X 75.0631,Y 92.6297,Z 127,A 47.2896,B 24.9389,C -1.8061,E1 25.0995,E2 398.6818} C_DIS
LIN {X 71.5313,Y 95.3835,Z 127,A 49.253,B 24.9392,C -1.801,E1 25.0952,E2 396.7375} C_DIS
LIN {X 68.5474,Y 97.5518,Z 127,A 51.7032,B 24.9368,C -1.8364,E1 25.0894,E2 394.2123} C_DIS
LIN {X 64.6392,Y 100.1827,Z 127,A 53.0507,B 24.9395,C -1.7965,E1 25.0865,E2 392.9635} C_DIS
LIN {X 59.9408,Y 103.0642,Z 127,A 55.8382,B 24.9388,C -1.807,E1 25.0798,E2 390.1599} C_DIS
LIN {X 56.9053,Y 104.7689,Z 127,A 57.5851,B 24.9384,C -1.8129,E1 25.0755,E2 388.4042} C_DIS
LIN {X 53.8283,Y 106.3836,Z 127,A 59.3341,B 24.938,C -1.8188,E1 25.0712,E2 386.646} C_DIS
LIN {X 50.3672,Y 108.0642,Z 127,A 61.0887,B 24.9381,C -1.8166,E1 25.0668,E2 384.9011} C_DIS
LIN {X 47.3235,Y 109.4319,Z 127,A 62.6627,B 24.9381,C -1.817,E1 25.0627,E2 383.33} C_DIS
LIN {X 43.5307,Y 110.9946,Z 127,A 64.4029,B 24.9387,C -1.8084,E1 25.0583,E2 381.6143} C_DIS
LIN {X 40.7163,Y 112.0577,Z 127,A 66.0334,B 24.938,C -1.8183,E1 25.054,E2 379.9637} C_DIS
LIN {X 38.3175,Y 112.9006,Z 127,A 67.3587,B 24.9376,C -1.8242,E1 25.0505,E2 378.6272} C_DIS
LIN {X 31.8342,Y 114.8991,Z 127,A 70.488,B 24.9379,C -1.8205,E1 25.0421,E2 375.5121} C_DIS
LIN {X 27.9287,Y 115.9087,Z 127,A 72.514,B 24.9375,C -1.8257,E1 25.0366,E2 373.4768} C_DIS
LIN {X 24.3689,Y 116.7092,Z 127,A 74.3283,B 24.9373,C -1.8294,E1 25.0317,E2 371.6561} C_DIS
LIN {X 21.196,Y 117.3263,Z 127,A 75.8354,B 24.9373,C -1.8279,E1 25.0275,E2 370.1542} C_DIS
LIN {X 17.5331,Y 117.9313,Z 127,A 77.75,B 24.9369,C -1.8344,E1 25.0222,E2 368.2261} C_DIS
LIN {X 13.8852,Y 118.4142,Z 127,A 79.7086,B 24.9363,C -1.8435,E1 25.0167,E2 366.2473} C_DIS
LIN {X 9.496,Y 118.8468,Z 127,A 81.5138,B 24.9373,C -1.8293,E1 25.0118,E2 364.4768} C_DIS
LIN {X 6.3998,Y 119.0538,Z 127,A 83.0647,B 24.9371,C -1.832,E1 25.0075,E2 362.9201} C_DIS
LIN {X 1.7684,Y 119.2132,Z 127,A 85.5669,B 24.9362,C -1.8443,E1 25.0004,E2 360.3893} C_DIS
LIN {X -1.5612,Y 119.217,Z 127,A 86.7346,B 24.9376,C -1.8243,E1 24.9973,E2 359.2689} C_DIS
LIN {X -4.0958,Y 119.156,Z 127,A 88.0393,B 24.9374,C -1.8278,E1 24.9936,E2 357.9557} C_DIS
LIN {X -9.7066,Y 118.8299,Z 127,A 90.6501,B 24.9377,C -1.8227,E1 24.9864,E2 355.3562} C_DIS
LIN {X -14.4654,Y 118.3463,Z 127,A 93.1604,B 24.9372,C -1.8309,E1 24.9793,E2 352.8249} C_DIS
LIN {X -18.489,Y 117.7835,Z 127,A 94.9899,B 24.9376,C -1.8241,E1 24.9743,E2 351.01} C_DIS
LIN {X -21.2445,Y 117.3176,Z 127,A 96.3282,B 24.9377,C -1.8229,E1 24.9706,E2 349.6733} C_DIS
LIN {X -24.1477,Y 116.7546,Z 127,A 97.7249,B 24.9379,C -1.8206,E1 24.9668,E2 348.2805} C_DIS
LIN {X -27.2921,Y 116.0607,Z 127,A 99.4078,B 24.9376,C -1.8252,E1 24.9622,E2 346.5845} C_DIS
LIN {X -33.8504,Y 114.3192,Z 127,A 102.5686,B 24.9381,C -1.8173,E1 24.9538,E2 343.4375} C_DIS
LIN {X -36.9149,Y 113.367,Z 127,A 104.1769,B 24.9381,C -1.8184,E1 24.9494,E2 341.8237} C_DIS
LIN {X -44.933,Y 110.4344,Z 127,A 108.2877,B 24.9384,C -1.8132,E1 24.9387,E2 337.7167} C_DIS
LIN {X -48.2102,Y 109.0453,Z 127,A 109.9229,B 24.9388,C -1.8073,E1 24.9345,E2 336.0916} C_DIS
LIN {X -53.0485,Y 106.7736,Z 127,A 112.9913,B 24.9376,C -1.8252,E1 24.9267,E2 332.9728} C_DIS
LIN {X -56.4087,Y 105.0383,Z 127,A 115.02,B 24.9371,C -1.8313,E1 24.9217,E2 330.9237} C_DIS
LIN {X -60.4363,Y 102.7728,Z 127,A 117.1117,B 24.9378,C -1.8216,E1 24.9167,E2 328.8488} C_DIS
LIN {X -63.9242,Y 100.6417,Z 127,A 118.4548,B 24.9399,C -1.7908,E1 24.9137,E2 327.5749} C_DIS
LIN {X -66.9519,Y 98.6519,Z 127,A 121.0062,B 24.9377,C -1.8226,E1 24.9076,E2 324.9391} C_DIS
LIN {X -70.9526,Y 95.8168,Z 127,A 122.6425,B 24.9402,C -1.7863,E1 24.9041,E2 323.3835} C_DIS
LIN {X -75.0527,Y 92.6381,Z 127,A 125.1856,B 24.9404,C -1.7831,E1 24.8985,E2 320.8387} C_DIS
LIN {X -77.5773,Y 90.5351,Z 127,A 127.2457,B 24.9393,C -1.8003,E1 24.894,E2 318.7297} C_DIS
LIN {X -80.4228,Y 88.0168,Z 127,A 128.5267,B 24.9411,C -1.7725,E1 24.8915,E2 317.5097} C_DIS
LIN {X -84.5579,Y 84.0525,Z 127,A 131.1802,B 24.9418,C -1.7616,E1 24.8862,E2 314.8712} C_DIS
LIN {X -86.2871,Y 82.278,Z 127,A 133.1463,B 24.9398,C -1.7919,E1 24.8822,E2 312.8244} C_DIS
LIN {X -89.1523,Y 79.1633,Z 127,A 134.3046,B 24.9427,C -1.7491,E1 24.8802,E2 311.7627} C_DIS
LIN {X -92.4718,Y 75.258,Z 127,A 136.8427,B 24.9429,C -1.7458,E1 24.8757,E2 309.2209} C_DIS
LIN {X -96.1527,Y 70.4939,Z 127,A 140.0026,B 24.9427,C -1.7493,E1 24.8703,E2 306.0378} C_DIS
LIN {X -98.3444,Y 67.4046,Z 127,A 141.9902,B 24.9425,C -1.7513,E1 24.867,E2 304.0356} C_DIS
LIN {X -100.4348,Y 64.2465,Z 127,A 143.6898,B 24.9432,C -1.741,E1 24.8645,E2 302.3519} C_DIS
LIN {X -103.4847,Y 59.2089,Z 127,A 146.4936,B 24.9438,C -1.7316,E1 24.8605,E2 299.556} C_DIS
LIN {X -106.118,Y 54.3481,Z 127,A 148.8758,B 24.9451,C -1.7121,E1 24.8574,E2 297.2077} C_DIS
LIN {X -108.7761,Y 48.8112,Z 127,A 151.9211,B 24.9454,C -1.7071,E1 24.8537,E2 294.1579} C_DIS
LIN {X -109.8478,Y 46.3486,Z 127,A 153.4729,B 24.9449,C -1.7141,E1 24.852,E2 292.5807} C_DIS
LIN {X -111.2243,Y 42.946,Z 127,A 156.3787,B 24.9421,C -1.7573,E1 24.849,E2 289.5555} C_DIS
LIN {X -113.4934,Y 36.5241,Z 127,A 158.416,B 24.9462,C -1.6942,E1 24.8473,E2 287.657} C_DIS
LIN {X -114.2994,Y 33.9173,Z 127,A 159.8205,B 24.9462,C -1.694,E1 24.8461,E2 286.245} C_DIS
LIN {X -115.3637,Y 30.1022,Z 127,A 161.8717,B 24.9462,C -1.6941,E1 24.8446,E2 284.1816} C_DIS
LIN {X -116.2183,Y 26.6097,Z 127,A 163.4337,B 24.947,C -1.6816,E1 24.8436,E2 282.6404} C_DIS
LIN {X -116.8546,Y 23.6606,Z 127,A 164.9353,B 24.9472,C -1.679,E1 24.8428,E2 281.1359} C_DIS
LIN {X -117.4225,Y 20.6612,Z 127,A 166.5811,B 24.947,C -1.6818,E1 24.842,E2 279.4737} C_DIS
LIN {X -118.0649,Y 16.5964,Z 127,A 168.4659,B 24.9476,C -1.6715,E1 24.8412,E2 277.6024} C_DIS
LIN {X -118.5614,Y 12.5675,Z 127,A 170.4533,B 24.9479,C -1.6666,E1 24.8405,E2 275.6145} C_DIS
LIN {X -118.8867,Y 8.9964,Z 127,A 172.1401,B 24.9484,C -1.6595,E1 24.8402,E2 273.9348} C_DIS
LIN {X -119.107,Y 5.3199,Z 127,A 173.9989,B 24.9485,C -1.6574,E1 24.8399,E2 272.0696} C_DIS
LIN {X -119.2123,Y 1.8188,Z 127,A 175.58,B 24.9491,C -1.6476,E1 24.8398,E2 270.5025} C_DIS
LIN {X -119.2112,Y -1.8769,Z 127,A 177.4475,B 24.9493,C -1.6457,E1 24.8398,E2 268.6283} C_DIS
LIN {X -119.1127,Y -5.186,Z 127,A 178.9817,B 24.9497,C -1.6381,E1 24.84,E2 267.1028} C_DIS
LIN {X -118.9232,Y -8.4977,Z 127,A -179.2562,B 24.9496,C -1.64,E1 24.8403,E2 265.3255} C_DIS
LIN {X -118.5882,Y -12.3116,Z 127,A -177.5496,B 24.9503,C -1.6285,E1 24.8408,E2 263.6363} C_DIS
LIN {X -118.2249,Y -15.415,Z 127,A -175.9818,B 24.9504,C -1.6265,E1 24.8413,E2 262.064} C_DIS
LIN {X -116.8804,Y -23.5354,Z 127,A -172.2015,B 24.9517,C -1.6063,E1 24.8431,E2 258.3092} C_DIS
LIN {X -116.1045,Y -27.1027,Z 127,A -169.6342,B 24.9499,C -1.6355,E1 24.8448,E2 255.6573} C_DIS
LIN {X -114.9709,Y -31.5701,Z 127,A -168.0873,B 24.952,C -1.6001,E1 24.8458,E2 254.1858} C_DIS
Enddeposition()
END
